// TIA Portal V16 export
// export: Created 2023-03-29T11:03:18.3037804Z, ExportSetting WithDefaults, DisplayName Totally Integrated Automation Portal, DisplayVersion V16 Update 6, DisplayName TIA Portal Version Control Interface, DisplayVersion V16 Update 2, DisplayName TIA Portal Openness, DisplayVersion V16 Update 6, DisplayName STEP 7 Professional, DisplayVersion V16 Update 6, DisplayName STEP 7 Safety, DisplayVersion V16, DisplayName WinCC Advanced, DisplayVersion V16 Update 6
ORGANIZATION_BLOCK "Main"   // OB1, LAD, ProgramCycle
TITLE = "Main Program Sweep (Cycle)"
{ S7_Optimized_Access := 'TRUE' }
VERSION : 0.1
// stored: AutoNumber true, IsIECCheckEnabled false, SetENOAutomatically false
   VAR_INPUT
      Initial_Call : Bool;   // Initial call of this OB
      Remanence : Bool;   // =True, if remanent data are available
   END_VAR
   VAR_TEMP   // added for the SCL form of the ladder/FBD networks
      _w1 : Bool;
      _w2 : Bool;
   END_VAR
BEGIN

REGION Network 1: Diagnostyka przerwań
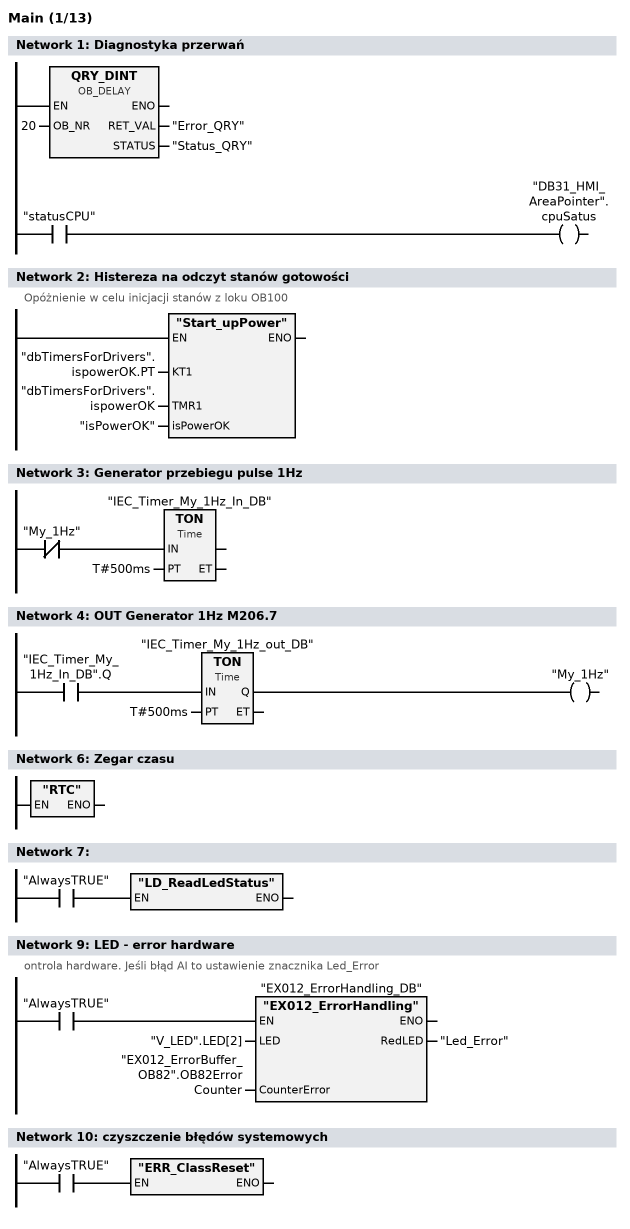
   RUNG wire#powerrail
      { S7_Templates := "obnr_type := OB_DELAY" } QRY_DINT(OB_NR := 20, RET_VAL => "Error_QRY", STATUS => "Status_QRY")
   END_RUNG
   RUNG wire#powerrail
      Contact( "statusCPU" )
      Coil( "DB31_HMI_AreaPointer".cpuSatus )
   END_RUNG
   // the same network as SCL:
   "Error_QRY" := QRY_DINT(OB_NR := 20, STATUS => "Status_QRY");
   "DB31_HMI_AreaPointer".cpuSatus := "statusCPU";
END_REGION

REGION Network 2: Histereza na odczyt stanów gotowości
   // Opóżnienie w celu inicjacji stanów z loku OB100
   RUNG wire#powerrail
      "Start_upPower"(KT1 := "dbTimersForDrivers".ispowerOK.PT, TMR1 := "dbTimersForDrivers".ispowerOK, isPowerOK := "isPowerOK")
   END_RUNG
   // the same network as SCL:
   "Start_upPower"(KT1 := "dbTimersForDrivers".ispowerOK.PT,
                   TMR1 := "dbTimersForDrivers".ispowerOK,
                   isPowerOK := "isPowerOK");
END_REGION

REGION Network 3: Generator przebiegu pulse 1Hz
   RUNG wire#powerrail
      I_Contact( "My_1Hz" )
      { S7_Templates := "time_type := Time" } "IEC_Timer_My_1Hz_In_DB".TON(pt := T#500ms, et =>)
   END_RUNG
   // the same network as SCL:
   "IEC_Timer_My_1Hz_In_DB".TON(IN := NOT "My_1Hz", PT := T#500ms);
END_REGION

REGION Network 4: OUT Generator 1Hz M206.7
   RUNG wire#powerrail
      Contact( "IEC_Timer_My_1Hz_In_DB".Q )
      { S7_Templates := "time_type := Time" } "IEC_Timer_My_1Hz_out_DB".TON(pt := T#500ms, et =>)
      Coil( "My_1Hz" )
   END_RUNG
   // the same network as SCL:
   "IEC_Timer_My_1Hz_out_DB".TON(IN := "IEC_Timer_My_1Hz_In_DB".Q, PT := T#500ms);
   "My_1Hz" := "IEC_Timer_My_1Hz_out_DB".Q;
END_REGION

REGION Network 6: Zegar czasu
   RUNG wire#powerrail
      "RTC"()
   END_RUNG
   // the same network as SCL:
   "RTC"();
END_REGION

REGION Network 7
   RUNG wire#powerrail
      Contact( "AlwaysTRUE" )
      "LD_ReadLedStatus"()
   END_RUNG
   // the same network as SCL:
   IF "AlwaysTRUE" THEN "LD_ReadLedStatus"(); END_IF;
END_REGION

REGION Network 8 (SCL): LED kontrola RUN
   // Przekazanie  stanu LED 1 CPU
   "DB31_HMI_AreaPointer".getPLCMode := "V_LED".LED[1];
END_REGION

REGION Network 9: LED - error hardware
   // ontrola hardware. Jeśli błąd AI to ustawienie znacznika Led_Error
   RUNG wire#powerrail
      Contact( "AlwaysTRUE" )
      "EX012_ErrorHandling_DB"(LED := "V_LED".LED[2], CounterError := "EX012_ErrorBuffer_OB82".OB82ErrorCounter, RedLED => "Led_Error")
   END_RUNG
   // the same network as SCL:
   IF "AlwaysTRUE" THEN
       "EX012_ErrorHandling_DB"(LED := "V_LED".LED[2],   // "EX012_ErrorHandling"
                               CounterError := "EX012_ErrorBuffer_OB82".OB82ErrorCounter,
                               RedLED => "Led_Error");
   END_IF;
END_REGION

REGION Network 10: czyszczenie błędów systemowych
   RUNG wire#powerrail
      Contact( "AlwaysTRUE" )
      "ERR_ClassReset"()
   END_RUNG
   // the same network as SCL:
   IF "AlwaysTRUE" THEN "ERR_ClassReset"(); END_IF;
END_REGION

REGION Network 11: kontrola błedów
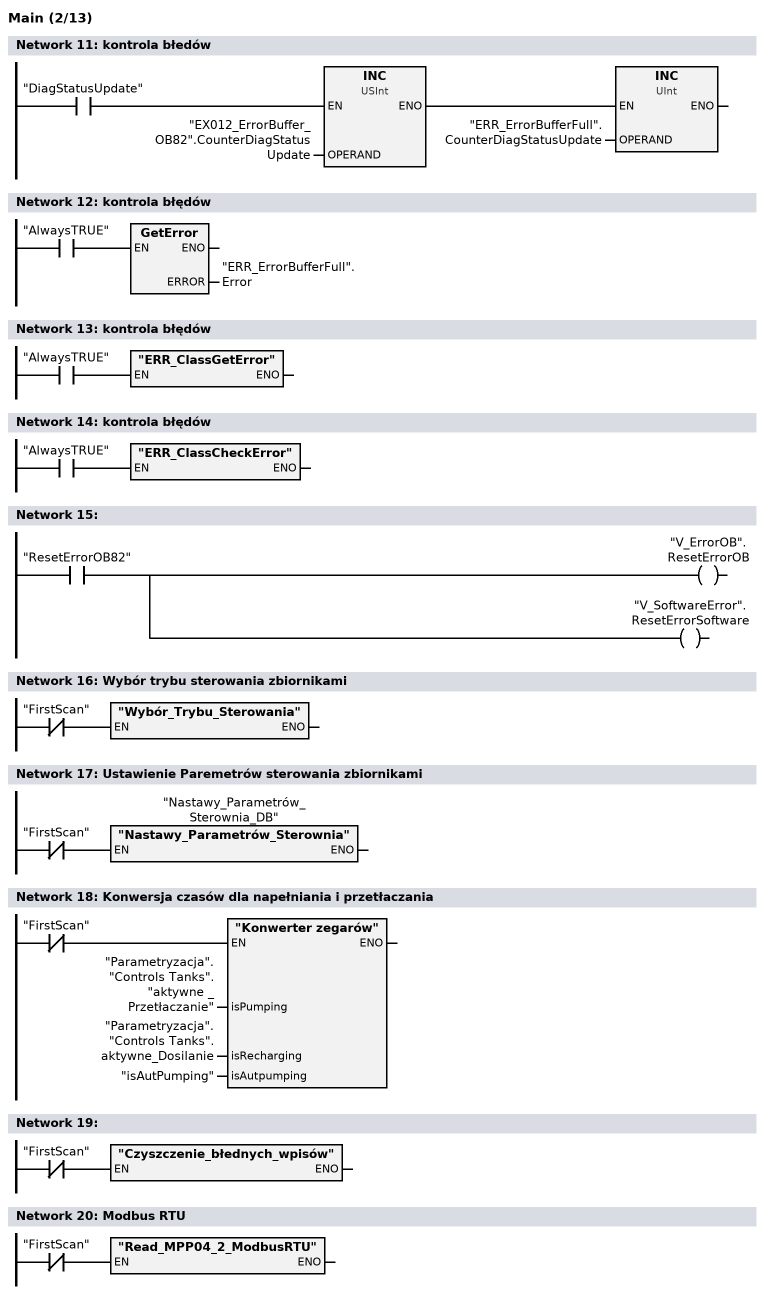
   RUNG wire#powerrail
      Contact( "DiagStatusUpdate" )
      { S7_Templates := "DestType := USInt" } Inc( "EX012_ErrorBuffer_OB82".CounterDiagStatusUpdate )
      { S7_Templates := "DestType := UInt" } Inc( "ERR_ErrorBufferFull".CounterDiagStatusUpdate )
   END_RUNG
   // the same network as SCL:
   IF "DiagStatusUpdate" THEN
       "EX012_ErrorBuffer_OB82".CounterDiagStatusUpdate := "EX012_ErrorBuffer_OB82".CounterDiagStatusUpdate + 1;
       "ERR_ErrorBufferFull".CounterDiagStatusUpdate := "ERR_ErrorBufferFull".CounterDiagStatusUpdate + 1;
   END_IF;
END_REGION

REGION Network 12: kontrola błędów
   // no SCL statement known for GetError: written as a call
   IF "AlwaysTRUE" THEN GetError(error => "ERR_ErrorBufferFull".Error); END_IF;
END_REGION

REGION Network 13: kontrola błędów
   RUNG wire#powerrail
      Contact( "AlwaysTRUE" )
      "ERR_ClassGetError"()
   END_RUNG
   // the same network as SCL:
   IF "AlwaysTRUE" THEN "ERR_ClassGetError"(); END_IF;
END_REGION

REGION Network 14: kontrola błędów
   RUNG wire#powerrail
      Contact( "AlwaysTRUE" )
      "ERR_ClassCheckError"()
   END_RUNG
   // the same network as SCL:
   IF "AlwaysTRUE" THEN "ERR_ClassCheckError"(); END_IF;
END_REGION

REGION Network 15
   RUNG wire#powerrail
      Contact( "ResetErrorOB82" )
      wire#w1
      Coil( "V_ErrorOB".ResetErrorOB )
   END_RUNG
   RUNG wire#w1
      Coil( "V_SoftwareError".ResetErrorSoftware )
   END_RUNG
   // the same network as SCL:
   "V_ErrorOB".ResetErrorOB := "ResetErrorOB82";
   "V_SoftwareError".ResetErrorSoftware := "ResetErrorOB82";
END_REGION

REGION Network 16: Wybór trybu sterowania zbiornikami
   RUNG wire#powerrail
      I_Contact( "FirstScan" )
      "Wybór_Trybu_Sterowania"()
   END_RUNG
   // the same network as SCL:
   IF NOT "FirstScan" THEN "Wybór_Trybu_Sterowania"(); END_IF;
END_REGION

REGION Network 17: Ustawienie Paremetrów sterowania zbiornikami
   RUNG wire#powerrail
      I_Contact( "FirstScan" )
      "Nastawy_Parametrów_Sterownia_DB"()
   END_RUNG
   // the same network as SCL:
   IF NOT "FirstScan" THEN
       "Nastawy_Parametrów_Sterownia_DB"();   // "Nastawy_Parametrów_Sterownia"
   END_IF;
END_REGION

REGION Network 18: Konwersja czasów dla napełniania i przetłaczania
   RUNG wire#powerrail
      I_Contact( "FirstScan" )
      "Konwerter zegarów"(isPumping := "Parametryzacja"."Controls Tanks"."aktywne _Przetłaczanie", isRecharging := "Parametryzacja"."Controls Tanks".aktywne_Dosilanie, isAutpumping := "isAutPumping")
   END_RUNG
   // the same network as SCL:
   IF NOT "FirstScan" THEN
       "Konwerter zegarów"(isPumping := "Parametryzacja"."Controls Tanks"."aktywne _Przetłaczanie",
                           isRecharging := "Parametryzacja"."Controls Tanks".aktywne_Dosilanie,
                           isAutpumping := "isAutPumping");
   END_IF;
END_REGION

REGION Network 19
   RUNG wire#powerrail
      I_Contact( "FirstScan" )
      "Czyszczenie_błednych_wpisów"()
   END_RUNG
   // the same network as SCL:
   IF NOT "FirstScan" THEN "Czyszczenie_błednych_wpisów"(); END_IF;
END_REGION

REGION Network 20: Modbus RTU
   RUNG wire#powerrail
      I_Contact( "FirstScan" )
      "Read_MPP04_2_ModbusRTU"()
   END_RUNG
   // the same network as SCL:
   IF NOT "FirstScan" THEN "Read_MPP04_2_ModbusRTU"(); END_IF;
END_REGION

REGION Network 21: Analogi przekazanie do dbHold Modbus TCP
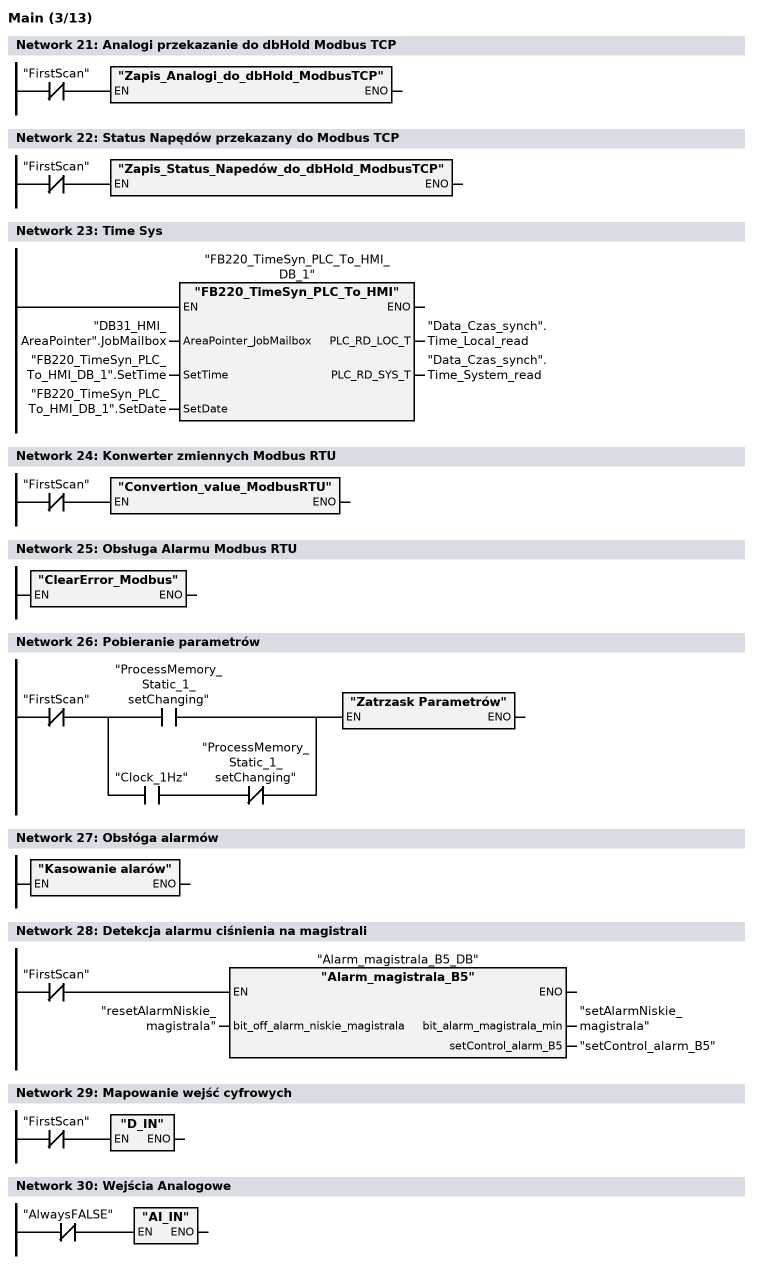
   RUNG wire#powerrail
      I_Contact( "FirstScan" )
      "Zapis_Analogi_do_dbHold_ModbusTCP"()
   END_RUNG
   // the same network as SCL:
   IF NOT "FirstScan" THEN "Zapis_Analogi_do_dbHold_ModbusTCP"(); END_IF;
END_REGION

REGION Network 22: Status Napędów przekazany do Modbus TCP
   RUNG wire#powerrail
      I_Contact( "FirstScan" )
      "Zapis_Status_Napedów_do_dbHold_ModbusTCP"()
   END_RUNG
   // the same network as SCL:
   IF NOT "FirstScan" THEN "Zapis_Status_Napedów_do_dbHold_ModbusTCP"(); END_IF;
END_REGION

REGION Network 23: Time Sys
   RUNG wire#powerrail
      "FB220_TimeSyn_PLC_To_HMI_DB_1"(AreaPointer_JobMailbox := "DB31_HMI_AreaPointer".JobMailbox, SetTime := "FB220_TimeSyn_PLC_To_HMI_DB_1".SetTime, SetDate := "FB220_TimeSyn_PLC_To_HMI_DB_1".SetDate, PLC_RD_LOC_T => "Data_Czas_synch".Time_Local_read, PLC_RD_SYS_T => "Data_Czas_synch".Time_System_read)
   END_RUNG
   // the same network as SCL:
   "FB220_TimeSyn_PLC_To_HMI_DB_1"(AreaPointer_JobMailbox := "DB31_HMI_AreaPointer".JobMailbox,   // "FB220_TimeSyn_PLC_To_HMI"
                           SetTime := "FB220_TimeSyn_PLC_To_HMI_DB_1".SetTime,
                           SetDate := "FB220_TimeSyn_PLC_To_HMI_DB_1".SetDate,
                           PLC_RD_LOC_T => "Data_Czas_synch".Time_Local_read,
                           PLC_RD_SYS_T => "Data_Czas_synch".Time_System_read);
END_REGION

REGION Network 24: Konwerter zmiennych Modbus RTU
   RUNG wire#powerrail
      I_Contact( "FirstScan" )
      "Convertion_value_ModbusRTU"()
   END_RUNG
   // the same network as SCL:
   IF NOT "FirstScan" THEN "Convertion_value_ModbusRTU"(); END_IF;
END_REGION

REGION Network 25: Obsługa Alarmu Modbus RTU
   RUNG wire#powerrail
      "ClearError_Modbus"()
   END_RUNG
   // the same network as SCL:
   "ClearError_Modbus"();
END_REGION

REGION Network 26: Pobieranie parametrów
   RUNG wire#powerrail
      I_Contact( "FirstScan" )
      wire#w1
      Contact( "ProcessMemory_Static_1_setChanging" )
      wire#w2
      "Zatrzask Parametrów"()
   END_RUNG
   RUNG wire#w1
      Contact( "Clock_1Hz" )
      I_Contact( "ProcessMemory_Static_1_setChanging" )
   END_RUNG wire#w2
   // the same network as SCL:
   IF NOT "FirstScan" AND ("ProcessMemory_Static_1_setChanging" OR ("Clock_1Hz" AND NOT "ProcessMemory_Static_1_setChanging")) THEN
       "Zatrzask Parametrów"();
   END_IF;
END_REGION

REGION Network 27: Obsłóga alarmów
   RUNG wire#powerrail
      "Kasowanie alarów"()
   END_RUNG
   // the same network as SCL:
   "Kasowanie alarów"();
END_REGION

REGION Network 28: Detekcja alarmu ciśnienia na magistrali
   RUNG wire#powerrail
      I_Contact( "FirstScan" )
      "Alarm_magistrala_B5_DB"(bit_off_alarm_niskie_magistrala := "resetAlarmNiskie_magistrala", bit_alarm_magistrala_min => "setAlarmNiskie_magistrala", setControl_alarm_B5 => "setControl_alarm_B5")
   END_RUNG
   // the same network as SCL:
   IF NOT "FirstScan" THEN
       "Alarm_magistrala_B5_DB"(bit_off_alarm_niskie_magistrala := "resetAlarmNiskie_magistrala",   // "Alarm_magistrala_B5"
                               bit_alarm_magistrala_min => "setAlarmNiskie_magistrala",
                               setControl_alarm_B5 => "setControl_alarm_B5");
   END_IF;
END_REGION

REGION Network 29: Mapowanie wejść cyfrowych
   RUNG wire#powerrail
      I_Contact( "FirstScan" )
      "D_IN"()
   END_RUNG
   // the same network as SCL:
   IF NOT "FirstScan" THEN "D_IN"(); END_IF;
END_REGION

REGION Network 30: Wejścia Analogowe
   RUNG wire#powerrail
      I_Contact( "AlwaysFALSE" )
      "AI_IN"()
   END_RUNG
   // the same network as SCL:
   IF NOT "AlwaysFALSE" THEN "AI_IN"(); END_IF;
END_REGION

REGION Network 31: Detekcja błędu nadajnika położenia Z10
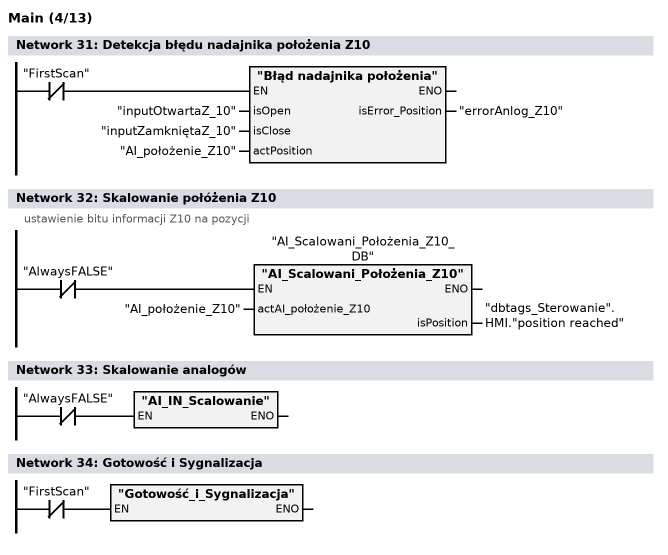
   RUNG wire#powerrail
      I_Contact( "FirstScan" )
      "Błąd nadajnika położenia"(isOpen := "inputOtwartaZ_10", isClose := "inputZamkniętaZ_10", actPosition := "AI_położenie_Z10", isError_Position => "errorAnlog_Z10")
   END_RUNG
   // the same network as SCL:
   IF NOT "FirstScan" THEN
       "Błąd nadajnika położenia"(isOpen := "inputOtwartaZ_10",
                               isClose := "inputZamkniętaZ_10",
                               actPosition := "AI_położenie_Z10",
                               isError_Position => "errorAnlog_Z10");
   END_IF;
END_REGION

REGION Network 32: Skalowanie połóżenia Z10
   // ustawienie bitu informacji Z10 na pozycji
   RUNG wire#powerrail
      I_Contact( "AlwaysFALSE" )
      "AI_Scalowani_Położenia_Z10_DB"(actAI_położenie_Z10 := "AI_położenie_Z10", isPosition => "dbtags_Sterowanie".HMI."position reached")
   END_RUNG
   // the same network as SCL:
   IF NOT "AlwaysFALSE" THEN
       "AI_Scalowani_Położenia_Z10_DB"(actAI_położenie_Z10 := "AI_położenie_Z10",   // "AI_Scalowani_Położenia_Z10"
                               isPosition => "dbtags_Sterowanie".HMI."position reached");
   END_IF;
END_REGION

REGION Network 33: Skalowanie analogów
   RUNG wire#powerrail
      I_Contact( "AlwaysFALSE" )
      "AI_IN_Scalowanie"()
   END_RUNG
   // the same network as SCL:
   IF NOT "AlwaysFALSE" THEN "AI_IN_Scalowanie"(); END_IF;
END_REGION

REGION Network 34: Gotowość i Sygnalizacja
   RUNG wire#powerrail
      I_Contact( "FirstScan" )
      "Gotowość_i_Sygnalizacja"()
   END_RUNG
   // the same network as SCL:
   IF NOT "FirstScan" THEN "Gotowość_i_Sygnalizacja"(); END_IF;
END_REGION

REGION Network 35
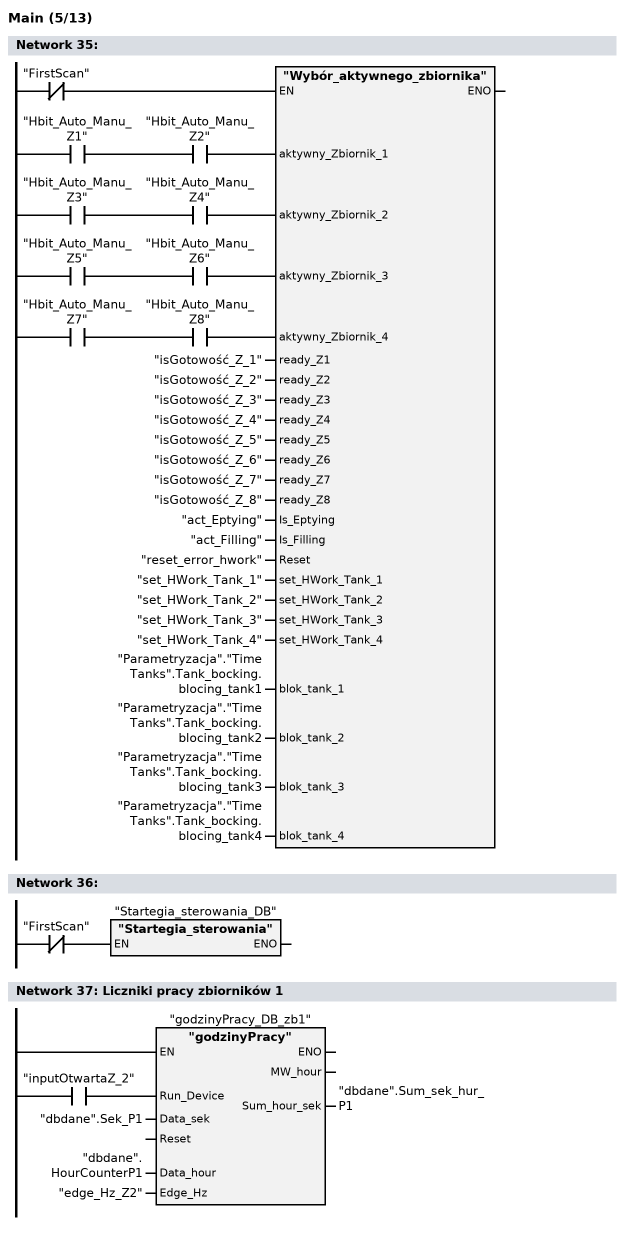
   RUNG wire#powerrail
      I_Contact( "FirstScan" )
      "Wybór_aktywnego_zbiornika"(aktywny_Zbiornik_1 := wire#w1, aktywny_Zbiornik_2 := wire#w2, aktywny_Zbiornik_3 := wire#w3, aktywny_Zbiornik_4 := wire#w4, ready_Z1 := "isGotowość_Z_1", ready_Z2 := "isGotowość_Z_2", ready_Z3 := "isGotowość_Z_3", ready_Z4 := "isGotowość_Z_4", ready_Z5 := "isGotowość_Z_5", ready_Z6 := "isGotowość_Z_6", ready_Z7 := "isGotowość_Z_7", ready_Z8 := "isGotowość_Z_8", Is_Eptying := "act_Eptying", Is_Filling := "act_Filling", Reset := "reset_error_hwork", set_HWork_Tank_1 := "set_HWork_Tank_1", set_HWork_Tank_2 := "set_HWork_Tank_2", set_HWork_Tank_3 := "set_HWork_Tank_3", set_HWork_Tank_4 := "set_HWork_Tank_4", blok_tank_1 := "Parametryzacja"."Time Tanks".Tank_bocking.blocing_tank1, blok_tank_2 := "Parametryzacja"."Time Tanks".Tank_bocking.blocing_tank2, blok_tank_3 := "Parametryzacja"."Time Tanks".Tank_bocking.blocing_tank3, blok_tank_4 := "Parametryzacja"."Time Tanks".Tank_bocking.blocing_tank4)
   END_RUNG
   RUNG wire#powerrail
      Contact( "Hbit_Auto_Manu_Z1" )
      Contact( "Hbit_Auto_Manu_Z2" )
   END_RUNG wire#w1
   RUNG wire#powerrail
      Contact( "Hbit_Auto_Manu_Z3" )
      Contact( "Hbit_Auto_Manu_Z4" )
   END_RUNG wire#w2
   RUNG wire#powerrail
      Contact( "Hbit_Auto_Manu_Z5" )
      Contact( "Hbit_Auto_Manu_Z6" )
   END_RUNG wire#w3
   RUNG wire#powerrail
      Contact( "Hbit_Auto_Manu_Z7" )
      Contact( "Hbit_Auto_Manu_Z8" )
   END_RUNG wire#w4
   // the same network as SCL:
   IF NOT "FirstScan" THEN
       "Wybór_aktywnego_zbiornika"(aktywny_Zbiornik_1 := "Hbit_Auto_Manu_Z1" AND "Hbit_Auto_Manu_Z2",
                               aktywny_Zbiornik_2 := "Hbit_Auto_Manu_Z3" AND "Hbit_Auto_Manu_Z4",
                               aktywny_Zbiornik_3 := "Hbit_Auto_Manu_Z5" AND "Hbit_Auto_Manu_Z6",
                               aktywny_Zbiornik_4 := "Hbit_Auto_Manu_Z7" AND "Hbit_Auto_Manu_Z8",
                               ready_Z1 := "isGotowość_Z_1",
                               ready_Z2 := "isGotowość_Z_2",
                               ready_Z3 := "isGotowość_Z_3",
                               ready_Z4 := "isGotowość_Z_4",
                               ready_Z5 := "isGotowość_Z_5",
                               ready_Z6 := "isGotowość_Z_6",
                               ready_Z7 := "isGotowość_Z_7",
                               ready_Z8 := "isGotowość_Z_8",
                               Is_Eptying := "act_Eptying",
                               Is_Filling := "act_Filling",
                               Reset := "reset_error_hwork",
                               set_HWork_Tank_1 := "set_HWork_Tank_1",
                               set_HWork_Tank_2 := "set_HWork_Tank_2",
                               set_HWork_Tank_3 := "set_HWork_Tank_3",
                               set_HWork_Tank_4 := "set_HWork_Tank_4",
                               blok_tank_1 := "Parametryzacja"."Time Tanks".Tank_bocking.blocing_tank1,
                               blok_tank_2 := "Parametryzacja"."Time Tanks".Tank_bocking.blocing_tank2,
                               blok_tank_3 := "Parametryzacja"."Time Tanks".Tank_bocking.blocing_tank3,
                               blok_tank_4 := "Parametryzacja"."Time Tanks".Tank_bocking.blocing_tank4);
   END_IF;
END_REGION

REGION Network 36
   RUNG wire#powerrail
      I_Contact( "FirstScan" )
      "Startegia_sterowania_DB"()
   END_RUNG
   // the same network as SCL:
   IF NOT "FirstScan" THEN
       "Startegia_sterowania_DB"();   // "Startegia_sterowania"
   END_IF;
END_REGION

REGION Network 37: Liczniki pracy zbiorników 1
   RUNG wire#powerrail
      "godzinyPracy_DB_zb1"(Run_Device := wire#w1, Data_sek := "dbdane".Sek_P1, Reset :=, Data_hour := "dbdane".HourCounterP1, Edge_Hz := "edge_Hz_Z2", MW_hour =>, Sum_hour_sek => "dbdane".Sum_sek_hur_P1)
   END_RUNG
   RUNG wire#powerrail
      Contact( "inputOtwartaZ_2" )
   END_RUNG wire#w1
   // the same network as SCL:
   "godzinyPracy_DB_zb1"(Run_Device := "inputOtwartaZ_2",   // "godzinyPracy"
                         Data_sek := "dbdane".Sek_P1,
                         Data_hour := "dbdane".HourCounterP1,
                         Edge_Hz := "edge_Hz_Z2",
                         Sum_hour_sek => "dbdane".Sum_sek_hur_P1);
END_REGION

REGION Network 38: Liczniki pracy zbiorników 2
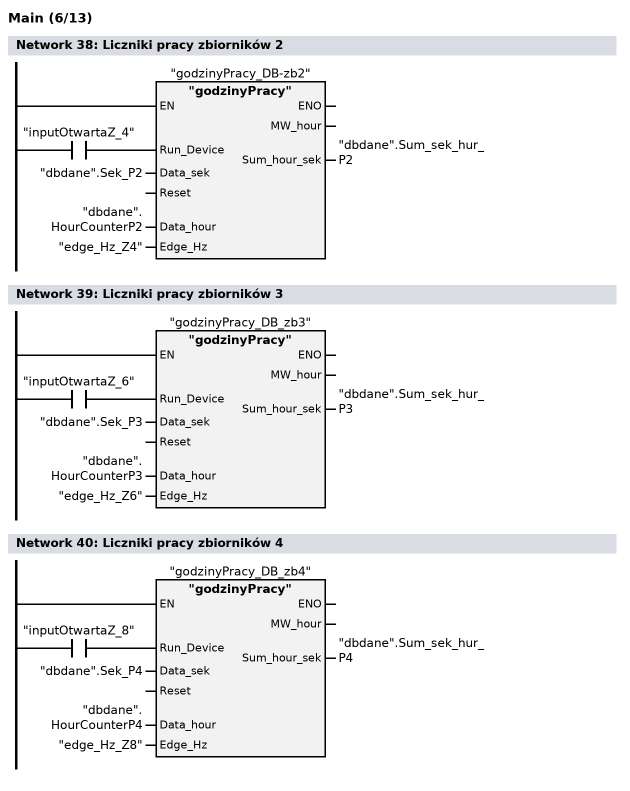
   RUNG wire#powerrail
      "godzinyPracy_DB-zb2"(Run_Device := wire#w1, Data_sek := "dbdane".Sek_P2, Reset :=, Data_hour := "dbdane".HourCounterP2, Edge_Hz := "edge_Hz_Z4", MW_hour =>, Sum_hour_sek => "dbdane".Sum_sek_hur_P2)
   END_RUNG
   RUNG wire#powerrail
      Contact( "inputOtwartaZ_4" )
   END_RUNG wire#w1
   // the same network as SCL:
   "godzinyPracy_DB-zb2"(Run_Device := "inputOtwartaZ_4",   // "godzinyPracy"
                         Data_sek := "dbdane".Sek_P2,
                         Data_hour := "dbdane".HourCounterP2,
                         Edge_Hz := "edge_Hz_Z4",
                         Sum_hour_sek => "dbdane".Sum_sek_hur_P2);
END_REGION

REGION Network 39: Liczniki pracy zbiorników 3
   RUNG wire#powerrail
      "godzinyPracy_DB_zb3"(Run_Device := wire#w1, Data_sek := "dbdane".Sek_P3, Reset :=, Data_hour := "dbdane".HourCounterP3, Edge_Hz := "edge_Hz_Z6", MW_hour =>, Sum_hour_sek => "dbdane".Sum_sek_hur_P3)
   END_RUNG
   RUNG wire#powerrail
      Contact( "inputOtwartaZ_6" )
   END_RUNG wire#w1
   // the same network as SCL:
   "godzinyPracy_DB_zb3"(Run_Device := "inputOtwartaZ_6",   // "godzinyPracy"
                         Data_sek := "dbdane".Sek_P3,
                         Data_hour := "dbdane".HourCounterP3,
                         Edge_Hz := "edge_Hz_Z6",
                         Sum_hour_sek => "dbdane".Sum_sek_hur_P3);
END_REGION

REGION Network 40: Liczniki pracy zbiorników 4
   RUNG wire#powerrail
      "godzinyPracy_DB_zb4"(Run_Device := wire#w1, Data_sek := "dbdane".Sek_P4, Reset :=, Data_hour := "dbdane".HourCounterP4, Edge_Hz := "edge_Hz_Z8", MW_hour =>, Sum_hour_sek => "dbdane".Sum_sek_hur_P4)
   END_RUNG
   RUNG wire#powerrail
      Contact( "inputOtwartaZ_8" )
   END_RUNG wire#w1
   // the same network as SCL:
   "godzinyPracy_DB_zb4"(Run_Device := "inputOtwartaZ_8",   // "godzinyPracy"
                         Data_sek := "dbdane".Sek_P4,
                         Data_hour := "dbdane".HourCounterP4,
                         Edge_Hz := "edge_Hz_Z8",
                         Sum_hour_sek => "dbdane".Sum_sek_hur_P4);
END_REGION

REGION Network 41: Sterowanie zbiornikami nr 1
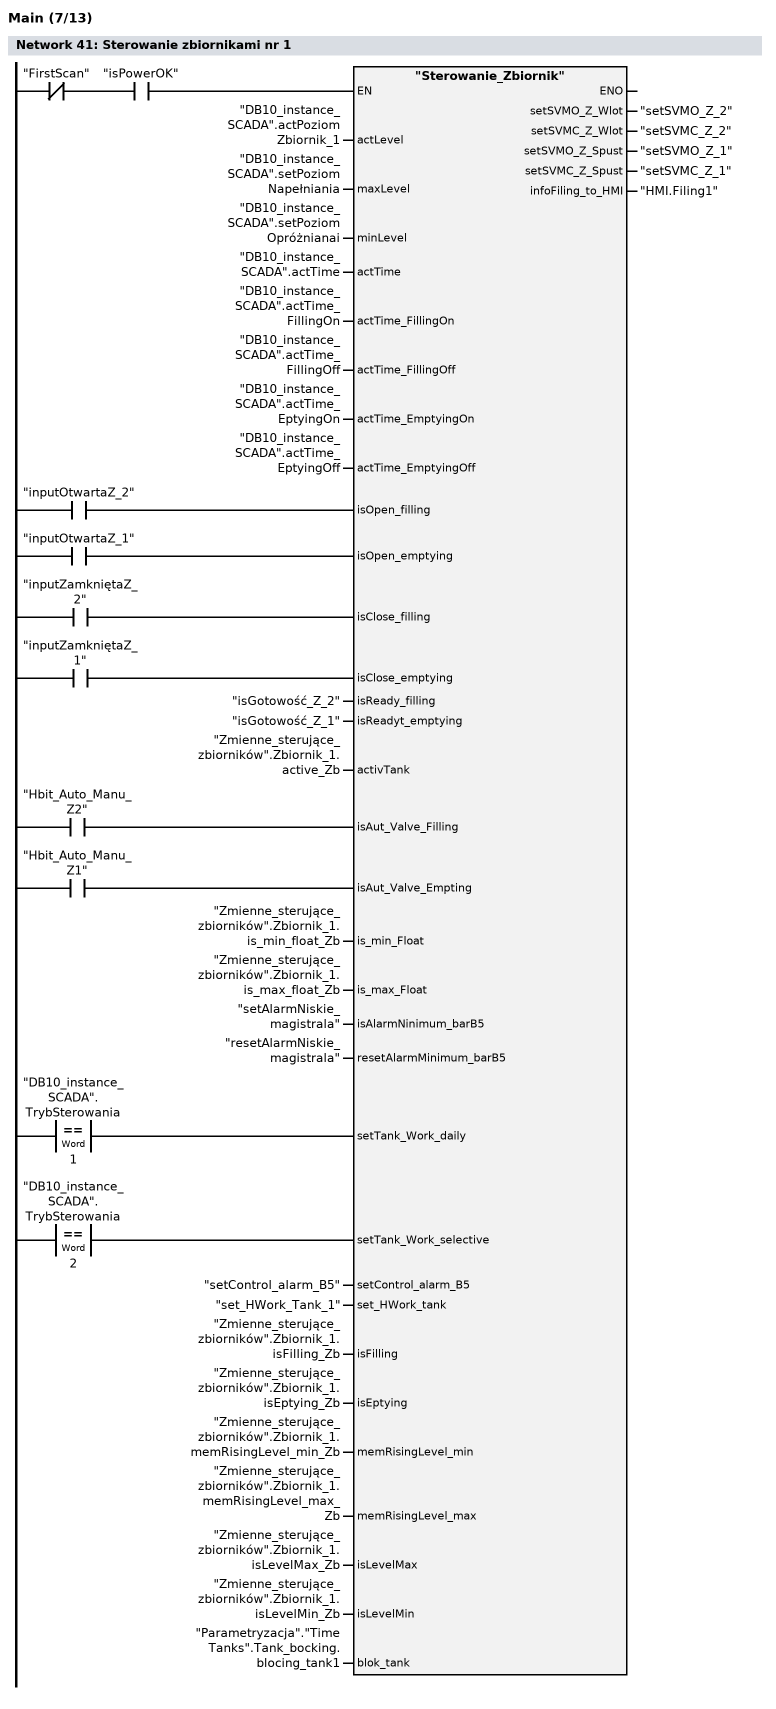
   RUNG wire#powerrail
      I_Contact( "FirstScan" )
      Contact( "isPowerOK" )
      "Sterowanie_Zbiornik"(isOpen_filling := wire#w1, isOpen_emptying := wire#w2, isClose_filling := wire#w3, isClose_emptying := wire#w4, isAut_Valve_Filling := wire#w5, isAut_Valve_Empting := wire#w6, setTank_Work_daily := wire#w7, setTank_Work_selective := wire#w8, actLevel := "DB10_instance_SCADA".actPoziomZbiornik_1, maxLevel := "DB10_instance_SCADA".setPoziomNapełniania, minLevel := "DB10_instance_SCADA".setPoziomOpróżnianai, actTime := "DB10_instance_SCADA".actTime, actTime_FillingOn := "DB10_instance_SCADA".actTime_FillingOn, actTime_FillingOff := "DB10_instance_SCADA".actTime_FillingOff, actTime_EmptyingOn := "DB10_instance_SCADA".actTime_EptyingOn, actTime_EmptyingOff := "DB10_instance_SCADA".actTime_EptyingOff, isReady_filling := "isGotowość_Z_2", isReadyt_emptying := "isGotowość_Z_1", activTank := "Zmienne_sterujące_zbiorników".Zbiornik_1.active_Zb, is_min_Float := "Zmienne_sterujące_zbiorników".Zbiornik_1.is_min_float_Zb, is_max_Float := "Zmienne_sterujące_zbiorników".Zbiornik_1.is_max_float_Zb, isAlarmNinimum_barB5 := "setAlarmNiskie_magistrala", resetAlarmMinimum_barB5 := "resetAlarmNiskie_magistrala", setControl_alarm_B5 := "setControl_alarm_B5", set_HWork_tank := "set_HWork_Tank_1", isFilling := "Zmienne_sterujące_zbiorników".Zbiornik_1.isFilling_Zb, isEptying := "Zmienne_sterujące_zbiorników".Zbiornik_1.isEptying_Zb, memRisingLevel_min := "Zmienne_sterujące_zbiorników".Zbiornik_1.memRisingLevel_min_Zb, memRisingLevel_max := "Zmienne_sterujące_zbiorników".Zbiornik_1.memRisingLevel_max_Zb, isLevelMax := "Zmienne_sterujące_zbiorników".Zbiornik_1.isLevelMax_Zb, isLevelMin := "Zmienne_sterujące_zbiorników".Zbiornik_1.isLevelMin_Zb, blok_tank := "Parametryzacja"."Time Tanks".Tank_bocking.blocing_tank1, setSVMO_Z_Wlot => "setSVMO_Z_2", setSVMC_Z_Wlot => "setSVMC_Z_2", setSVMO_Z_Spust => "setSVMO_Z_1", setSVMC_Z_Spust => "setSVMC_Z_1", infoFiling_to_HMI => "HMI.Filing1")
   END_RUNG
   RUNG wire#powerrail
      Contact( "inputOtwartaZ_2" )
   END_RUNG wire#w1
   RUNG wire#powerrail
      Contact( "inputOtwartaZ_1" )
   END_RUNG wire#w2
   RUNG wire#powerrail
      Contact( "inputZamkniętaZ_2" )
   END_RUNG wire#w3
   RUNG wire#powerrail
      Contact( "inputZamkniętaZ_1" )
   END_RUNG wire#w4
   RUNG wire#powerrail
      Contact( "Hbit_Auto_Manu_Z2" )
   END_RUNG wire#w5
   RUNG wire#powerrail
      Contact( "Hbit_Auto_Manu_Z1" )
   END_RUNG wire#w6
   RUNG wire#powerrail
      { S7_Templates := "SrcType := Word" } EQ_Contact(in1 := "DB10_instance_SCADA".TrybSterowania, in2 := 1)
   END_RUNG wire#w7
   RUNG wire#powerrail
      { S7_Templates := "SrcType := Word" } EQ_Contact(in1 := "DB10_instance_SCADA".TrybSterowania, in2 := 2)
   END_RUNG wire#w8
   // the same network as SCL:
   IF NOT "FirstScan" AND "isPowerOK" THEN
       "Sterowanie_Zbiornik"(actLevel := "DB10_instance_SCADA".actPoziomZbiornik_1,
                             maxLevel := "DB10_instance_SCADA".setPoziomNapełniania,
                             minLevel := "DB10_instance_SCADA".setPoziomOpróżnianai,
                             actTime := "DB10_instance_SCADA".actTime,
                             actTime_FillingOn := "DB10_instance_SCADA".actTime_FillingOn,
                             actTime_FillingOff := "DB10_instance_SCADA".actTime_FillingOff,
                             actTime_EmptyingOn := "DB10_instance_SCADA".actTime_EptyingOn,
                             actTime_EmptyingOff := "DB10_instance_SCADA".actTime_EptyingOff,
                             isOpen_filling := "inputOtwartaZ_2",
                             isOpen_emptying := "inputOtwartaZ_1",
                             isClose_filling := "inputZamkniętaZ_2",
                             isClose_emptying := "inputZamkniętaZ_1",
                             isReady_filling := "isGotowość_Z_2",
                             isReadyt_emptying := "isGotowość_Z_1",
                             activTank := "Zmienne_sterujące_zbiorników".Zbiornik_1.active_Zb,
                             isAut_Valve_Filling := "Hbit_Auto_Manu_Z2",
                             isAut_Valve_Empting := "Hbit_Auto_Manu_Z1",
                             is_min_Float := "Zmienne_sterujące_zbiorników".Zbiornik_1.is_min_float_Zb,
                             is_max_Float := "Zmienne_sterujące_zbiorników".Zbiornik_1.is_max_float_Zb,
                             isAlarmNinimum_barB5 := "setAlarmNiskie_magistrala",
                             resetAlarmMinimum_barB5 := "resetAlarmNiskie_magistrala",
                             setTank_Work_daily := "DB10_instance_SCADA".TrybSterowania = 1,
                             setTank_Work_selective := "DB10_instance_SCADA".TrybSterowania = 2,
                             setControl_alarm_B5 := "setControl_alarm_B5",
                             set_HWork_tank := "set_HWork_Tank_1",
                             isFilling := "Zmienne_sterujące_zbiorników".Zbiornik_1.isFilling_Zb,
                             isEptying := "Zmienne_sterujące_zbiorników".Zbiornik_1.isEptying_Zb,
                             memRisingLevel_min := "Zmienne_sterujące_zbiorników".Zbiornik_1.memRisingLevel_min_Zb,
                             memRisingLevel_max := "Zmienne_sterujące_zbiorników".Zbiornik_1.memRisingLevel_max_Zb,
                             isLevelMax := "Zmienne_sterujące_zbiorników".Zbiornik_1.isLevelMax_Zb,
                             isLevelMin := "Zmienne_sterujące_zbiorników".Zbiornik_1.isLevelMin_Zb,
                             blok_tank := "Parametryzacja"."Time Tanks".Tank_bocking.blocing_tank1,
                             setSVMO_Z_Wlot => "setSVMO_Z_2",
                             setSVMC_Z_Wlot => "setSVMC_Z_2",
                             setSVMO_Z_Spust => "setSVMO_Z_1",
                             setSVMC_Z_Spust => "setSVMC_Z_1",
                             infoFiling_to_HMI => "HMI.Filing1");
   END_IF;
END_REGION

REGION Network 42: Sterowanie zbiornikami nr 2
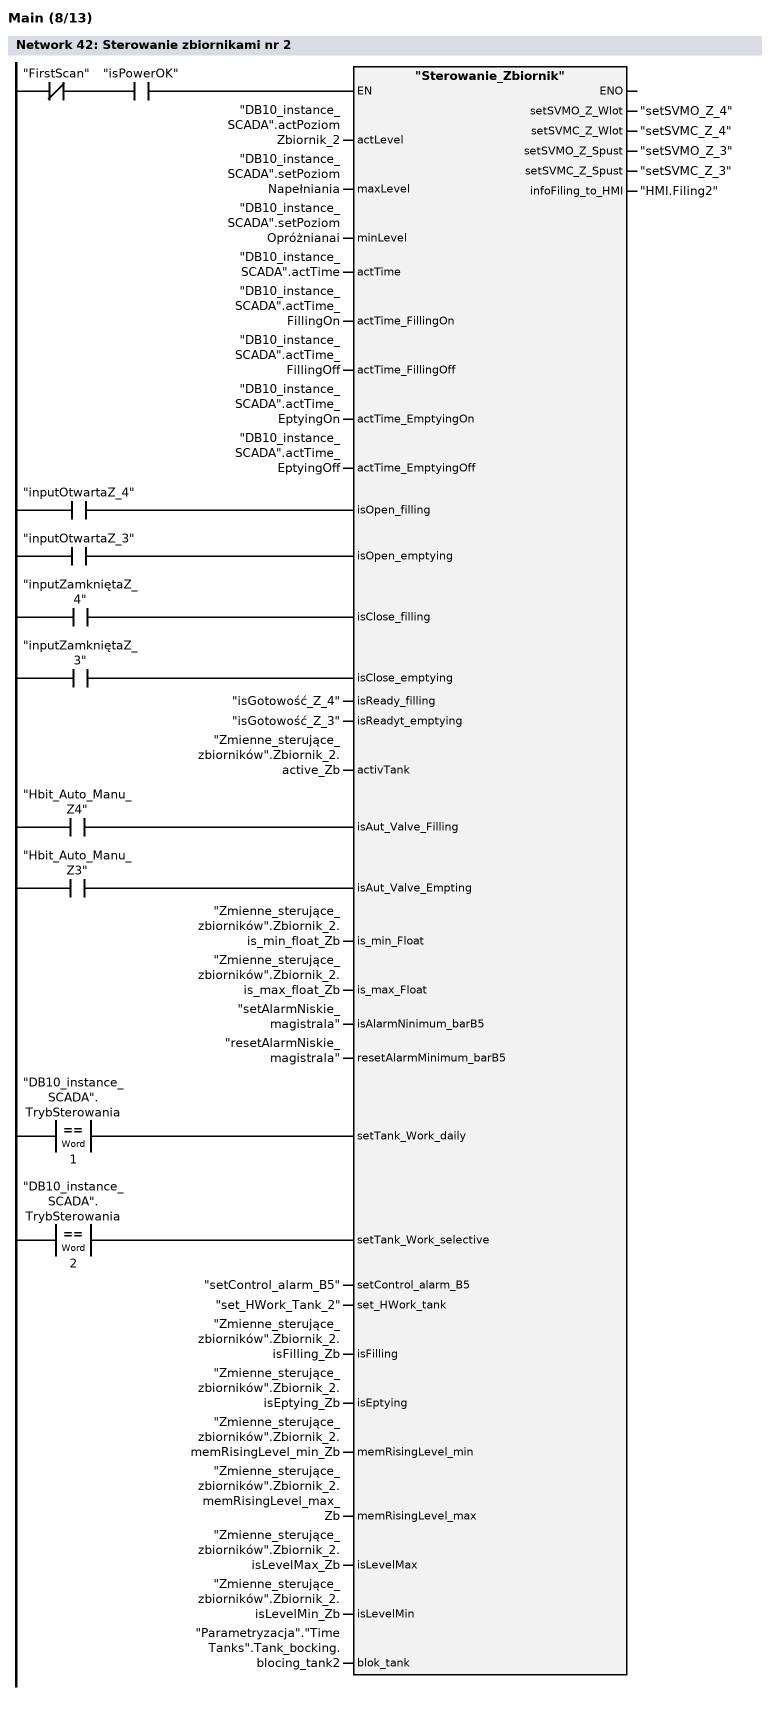
   RUNG wire#powerrail
      I_Contact( "FirstScan" )
      Contact( "isPowerOK" )
      "Sterowanie_Zbiornik"(isOpen_filling := wire#w1, isOpen_emptying := wire#w2, isClose_filling := wire#w3, isClose_emptying := wire#w4, isAut_Valve_Filling := wire#w5, isAut_Valve_Empting := wire#w6, setTank_Work_daily := wire#w7, setTank_Work_selective := wire#w8, actLevel := "DB10_instance_SCADA".actPoziomZbiornik_2, maxLevel := "DB10_instance_SCADA".setPoziomNapełniania, minLevel := "DB10_instance_SCADA".setPoziomOpróżnianai, actTime := "DB10_instance_SCADA".actTime, actTime_FillingOn := "DB10_instance_SCADA".actTime_FillingOn, actTime_FillingOff := "DB10_instance_SCADA".actTime_FillingOff, actTime_EmptyingOn := "DB10_instance_SCADA".actTime_EptyingOn, actTime_EmptyingOff := "DB10_instance_SCADA".actTime_EptyingOff, isReady_filling := "isGotowość_Z_4", isReadyt_emptying := "isGotowość_Z_3", activTank := "Zmienne_sterujące_zbiorników".Zbiornik_2.active_Zb, is_min_Float := "Zmienne_sterujące_zbiorników".Zbiornik_2.is_min_float_Zb, is_max_Float := "Zmienne_sterujące_zbiorników".Zbiornik_2.is_max_float_Zb, isAlarmNinimum_barB5 := "setAlarmNiskie_magistrala", resetAlarmMinimum_barB5 := "resetAlarmNiskie_magistrala", setControl_alarm_B5 := "setControl_alarm_B5", set_HWork_tank := "set_HWork_Tank_2", isFilling := "Zmienne_sterujące_zbiorników".Zbiornik_2.isFilling_Zb, isEptying := "Zmienne_sterujące_zbiorników".Zbiornik_2.isEptying_Zb, memRisingLevel_min := "Zmienne_sterujące_zbiorników".Zbiornik_2.memRisingLevel_min_Zb, memRisingLevel_max := "Zmienne_sterujące_zbiorników".Zbiornik_2.memRisingLevel_max_Zb, isLevelMax := "Zmienne_sterujące_zbiorników".Zbiornik_2.isLevelMax_Zb, isLevelMin := "Zmienne_sterujące_zbiorników".Zbiornik_2.isLevelMin_Zb, blok_tank := "Parametryzacja"."Time Tanks".Tank_bocking.blocing_tank2, setSVMO_Z_Wlot => "setSVMO_Z_4", setSVMC_Z_Wlot => "setSVMC_Z_4", setSVMO_Z_Spust => "setSVMO_Z_3", setSVMC_Z_Spust => "setSVMC_Z_3", infoFiling_to_HMI => "HMI.Filing2")
   END_RUNG
   RUNG wire#powerrail
      Contact( "inputOtwartaZ_4" )
   END_RUNG wire#w1
   RUNG wire#powerrail
      Contact( "inputOtwartaZ_3" )
   END_RUNG wire#w2
   RUNG wire#powerrail
      Contact( "inputZamkniętaZ_4" )
   END_RUNG wire#w3
   RUNG wire#powerrail
      Contact( "inputZamkniętaZ_3" )
   END_RUNG wire#w4
   RUNG wire#powerrail
      Contact( "Hbit_Auto_Manu_Z4" )
   END_RUNG wire#w5
   RUNG wire#powerrail
      Contact( "Hbit_Auto_Manu_Z3" )
   END_RUNG wire#w6
   RUNG wire#powerrail
      { S7_Templates := "SrcType := Word" } EQ_Contact(in1 := "DB10_instance_SCADA".TrybSterowania, in2 := 1)
   END_RUNG wire#w7
   RUNG wire#powerrail
      { S7_Templates := "SrcType := Word" } EQ_Contact(in1 := "DB10_instance_SCADA".TrybSterowania, in2 := 2)
   END_RUNG wire#w8
   // the same network as SCL:
   IF NOT "FirstScan" AND "isPowerOK" THEN
       "Sterowanie_Zbiornik"(actLevel := "DB10_instance_SCADA".actPoziomZbiornik_2,
                             maxLevel := "DB10_instance_SCADA".setPoziomNapełniania,
                             minLevel := "DB10_instance_SCADA".setPoziomOpróżnianai,
                             actTime := "DB10_instance_SCADA".actTime,
                             actTime_FillingOn := "DB10_instance_SCADA".actTime_FillingOn,
                             actTime_FillingOff := "DB10_instance_SCADA".actTime_FillingOff,
                             actTime_EmptyingOn := "DB10_instance_SCADA".actTime_EptyingOn,
                             actTime_EmptyingOff := "DB10_instance_SCADA".actTime_EptyingOff,
                             isOpen_filling := "inputOtwartaZ_4",
                             isOpen_emptying := "inputOtwartaZ_3",
                             isClose_filling := "inputZamkniętaZ_4",
                             isClose_emptying := "inputZamkniętaZ_3",
                             isReady_filling := "isGotowość_Z_4",
                             isReadyt_emptying := "isGotowość_Z_3",
                             activTank := "Zmienne_sterujące_zbiorników".Zbiornik_2.active_Zb,
                             isAut_Valve_Filling := "Hbit_Auto_Manu_Z4",
                             isAut_Valve_Empting := "Hbit_Auto_Manu_Z3",
                             is_min_Float := "Zmienne_sterujące_zbiorników".Zbiornik_2.is_min_float_Zb,
                             is_max_Float := "Zmienne_sterujące_zbiorników".Zbiornik_2.is_max_float_Zb,
                             isAlarmNinimum_barB5 := "setAlarmNiskie_magistrala",
                             resetAlarmMinimum_barB5 := "resetAlarmNiskie_magistrala",
                             setTank_Work_daily := "DB10_instance_SCADA".TrybSterowania = 1,
                             setTank_Work_selective := "DB10_instance_SCADA".TrybSterowania = 2,
                             setControl_alarm_B5 := "setControl_alarm_B5",
                             set_HWork_tank := "set_HWork_Tank_2",
                             isFilling := "Zmienne_sterujące_zbiorników".Zbiornik_2.isFilling_Zb,
                             isEptying := "Zmienne_sterujące_zbiorników".Zbiornik_2.isEptying_Zb,
                             memRisingLevel_min := "Zmienne_sterujące_zbiorników".Zbiornik_2.memRisingLevel_min_Zb,
                             memRisingLevel_max := "Zmienne_sterujące_zbiorników".Zbiornik_2.memRisingLevel_max_Zb,
                             isLevelMax := "Zmienne_sterujące_zbiorników".Zbiornik_2.isLevelMax_Zb,
                             isLevelMin := "Zmienne_sterujące_zbiorników".Zbiornik_2.isLevelMin_Zb,
                             blok_tank := "Parametryzacja"."Time Tanks".Tank_bocking.blocing_tank2,
                             setSVMO_Z_Wlot => "setSVMO_Z_4",
                             setSVMC_Z_Wlot => "setSVMC_Z_4",
                             setSVMO_Z_Spust => "setSVMO_Z_3",
                             setSVMC_Z_Spust => "setSVMC_Z_3",
                             infoFiling_to_HMI => "HMI.Filing2");
   END_IF;
END_REGION

REGION Network 43: Sterowanie zbiornikami nr 3
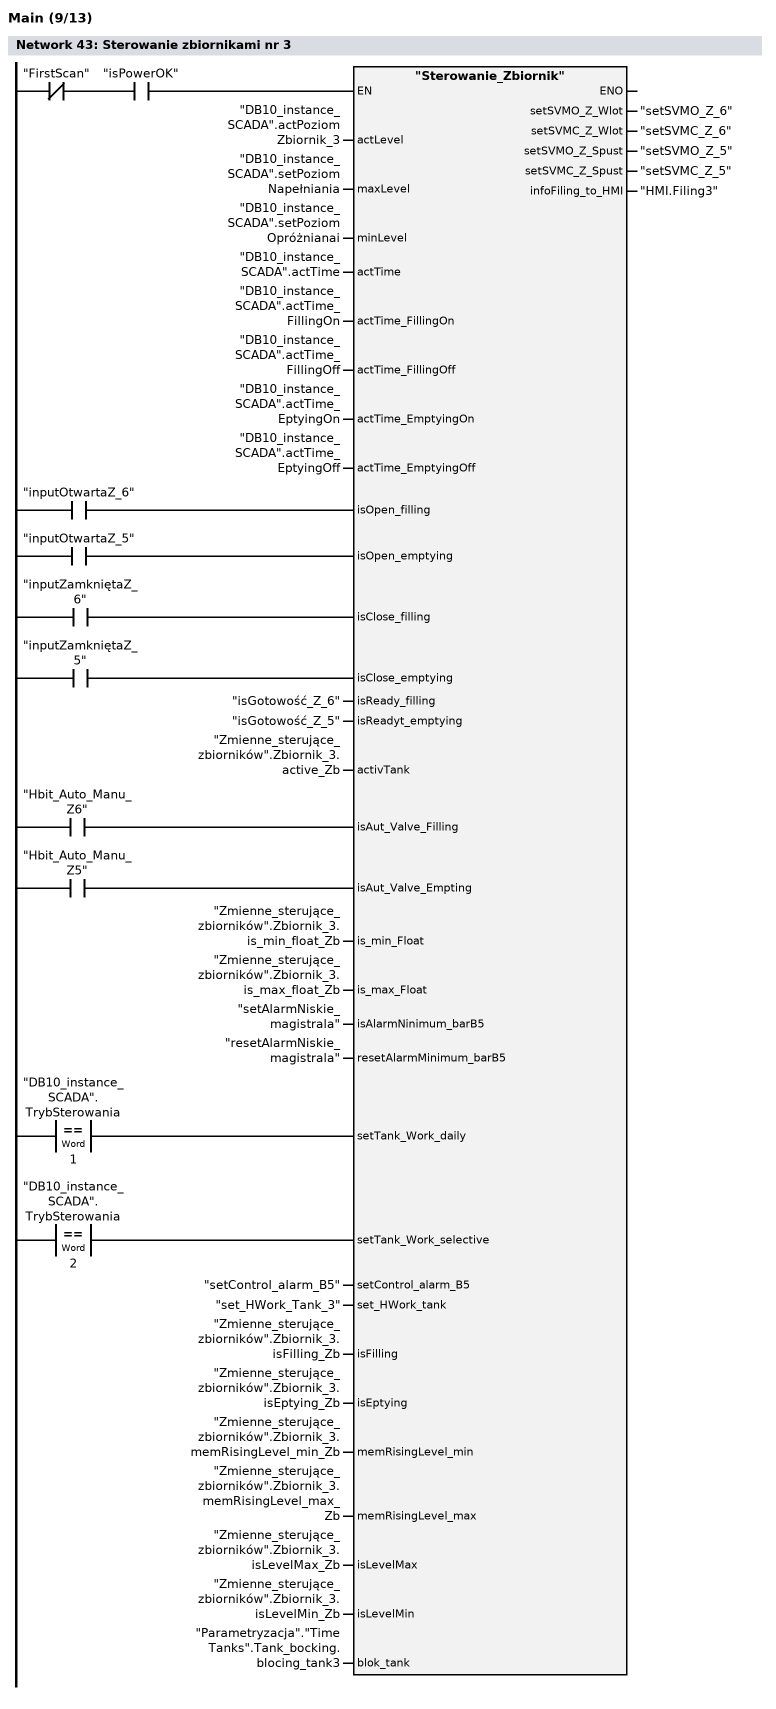
   RUNG wire#powerrail
      I_Contact( "FirstScan" )
      Contact( "isPowerOK" )
      "Sterowanie_Zbiornik"(isOpen_filling := wire#w1, isOpen_emptying := wire#w2, isClose_filling := wire#w3, isClose_emptying := wire#w4, isAut_Valve_Filling := wire#w5, isAut_Valve_Empting := wire#w6, setTank_Work_daily := wire#w7, setTank_Work_selective := wire#w8, actLevel := "DB10_instance_SCADA".actPoziomZbiornik_3, maxLevel := "DB10_instance_SCADA".setPoziomNapełniania, minLevel := "DB10_instance_SCADA".setPoziomOpróżnianai, actTime := "DB10_instance_SCADA".actTime, actTime_FillingOn := "DB10_instance_SCADA".actTime_FillingOn, actTime_FillingOff := "DB10_instance_SCADA".actTime_FillingOff, actTime_EmptyingOn := "DB10_instance_SCADA".actTime_EptyingOn, actTime_EmptyingOff := "DB10_instance_SCADA".actTime_EptyingOff, isReady_filling := "isGotowość_Z_6", isReadyt_emptying := "isGotowość_Z_5", activTank := "Zmienne_sterujące_zbiorników".Zbiornik_3.active_Zb, is_min_Float := "Zmienne_sterujące_zbiorników".Zbiornik_3.is_min_float_Zb, is_max_Float := "Zmienne_sterujące_zbiorników".Zbiornik_3.is_max_float_Zb, isAlarmNinimum_barB5 := "setAlarmNiskie_magistrala", resetAlarmMinimum_barB5 := "resetAlarmNiskie_magistrala", setControl_alarm_B5 := "setControl_alarm_B5", set_HWork_tank := "set_HWork_Tank_3", isFilling := "Zmienne_sterujące_zbiorników".Zbiornik_3.isFilling_Zb, isEptying := "Zmienne_sterujące_zbiorników".Zbiornik_3.isEptying_Zb, memRisingLevel_min := "Zmienne_sterujące_zbiorników".Zbiornik_3.memRisingLevel_min_Zb, memRisingLevel_max := "Zmienne_sterujące_zbiorników".Zbiornik_3.memRisingLevel_max_Zb, isLevelMax := "Zmienne_sterujące_zbiorników".Zbiornik_3.isLevelMax_Zb, isLevelMin := "Zmienne_sterujące_zbiorników".Zbiornik_3.isLevelMin_Zb, blok_tank := "Parametryzacja"."Time Tanks".Tank_bocking.blocing_tank3, setSVMO_Z_Wlot => "setSVMO_Z_6", setSVMC_Z_Wlot => "setSVMC_Z_6", setSVMO_Z_Spust => "setSVMO_Z_5", setSVMC_Z_Spust => "setSVMC_Z_5", infoFiling_to_HMI => "HMI.Filing3")
   END_RUNG
   RUNG wire#powerrail
      Contact( "inputOtwartaZ_6" )
   END_RUNG wire#w1
   RUNG wire#powerrail
      Contact( "inputOtwartaZ_5" )
   END_RUNG wire#w2
   RUNG wire#powerrail
      Contact( "inputZamkniętaZ_6" )
   END_RUNG wire#w3
   RUNG wire#powerrail
      Contact( "inputZamkniętaZ_5" )
   END_RUNG wire#w4
   RUNG wire#powerrail
      Contact( "Hbit_Auto_Manu_Z6" )
   END_RUNG wire#w5
   RUNG wire#powerrail
      Contact( "Hbit_Auto_Manu_Z5" )
   END_RUNG wire#w6
   RUNG wire#powerrail
      { S7_Templates := "SrcType := Word" } EQ_Contact(in1 := "DB10_instance_SCADA".TrybSterowania, in2 := 1)
   END_RUNG wire#w7
   RUNG wire#powerrail
      { S7_Templates := "SrcType := Word" } EQ_Contact(in1 := "DB10_instance_SCADA".TrybSterowania, in2 := 2)
   END_RUNG wire#w8
   // the same network as SCL:
   IF NOT "FirstScan" AND "isPowerOK" THEN
       "Sterowanie_Zbiornik"(actLevel := "DB10_instance_SCADA".actPoziomZbiornik_3,
                             maxLevel := "DB10_instance_SCADA".setPoziomNapełniania,
                             minLevel := "DB10_instance_SCADA".setPoziomOpróżnianai,
                             actTime := "DB10_instance_SCADA".actTime,
                             actTime_FillingOn := "DB10_instance_SCADA".actTime_FillingOn,
                             actTime_FillingOff := "DB10_instance_SCADA".actTime_FillingOff,
                             actTime_EmptyingOn := "DB10_instance_SCADA".actTime_EptyingOn,
                             actTime_EmptyingOff := "DB10_instance_SCADA".actTime_EptyingOff,
                             isOpen_filling := "inputOtwartaZ_6",
                             isOpen_emptying := "inputOtwartaZ_5",
                             isClose_filling := "inputZamkniętaZ_6",
                             isClose_emptying := "inputZamkniętaZ_5",
                             isReady_filling := "isGotowość_Z_6",
                             isReadyt_emptying := "isGotowość_Z_5",
                             activTank := "Zmienne_sterujące_zbiorników".Zbiornik_3.active_Zb,
                             isAut_Valve_Filling := "Hbit_Auto_Manu_Z6",
                             isAut_Valve_Empting := "Hbit_Auto_Manu_Z5",
                             is_min_Float := "Zmienne_sterujące_zbiorników".Zbiornik_3.is_min_float_Zb,
                             is_max_Float := "Zmienne_sterujące_zbiorników".Zbiornik_3.is_max_float_Zb,
                             isAlarmNinimum_barB5 := "setAlarmNiskie_magistrala",
                             resetAlarmMinimum_barB5 := "resetAlarmNiskie_magistrala",
                             setTank_Work_daily := "DB10_instance_SCADA".TrybSterowania = 1,
                             setTank_Work_selective := "DB10_instance_SCADA".TrybSterowania = 2,
                             setControl_alarm_B5 := "setControl_alarm_B5",
                             set_HWork_tank := "set_HWork_Tank_3",
                             isFilling := "Zmienne_sterujące_zbiorników".Zbiornik_3.isFilling_Zb,
                             isEptying := "Zmienne_sterujące_zbiorników".Zbiornik_3.isEptying_Zb,
                             memRisingLevel_min := "Zmienne_sterujące_zbiorników".Zbiornik_3.memRisingLevel_min_Zb,
                             memRisingLevel_max := "Zmienne_sterujące_zbiorników".Zbiornik_3.memRisingLevel_max_Zb,
                             isLevelMax := "Zmienne_sterujące_zbiorników".Zbiornik_3.isLevelMax_Zb,
                             isLevelMin := "Zmienne_sterujące_zbiorników".Zbiornik_3.isLevelMin_Zb,
                             blok_tank := "Parametryzacja"."Time Tanks".Tank_bocking.blocing_tank3,
                             setSVMO_Z_Wlot => "setSVMO_Z_6",
                             setSVMC_Z_Wlot => "setSVMC_Z_6",
                             setSVMO_Z_Spust => "setSVMO_Z_5",
                             setSVMC_Z_Spust => "setSVMC_Z_5",
                             infoFiling_to_HMI => "HMI.Filing3");
   END_IF;
END_REGION

REGION Network 44: Sterowanie zbiornikami nr 4
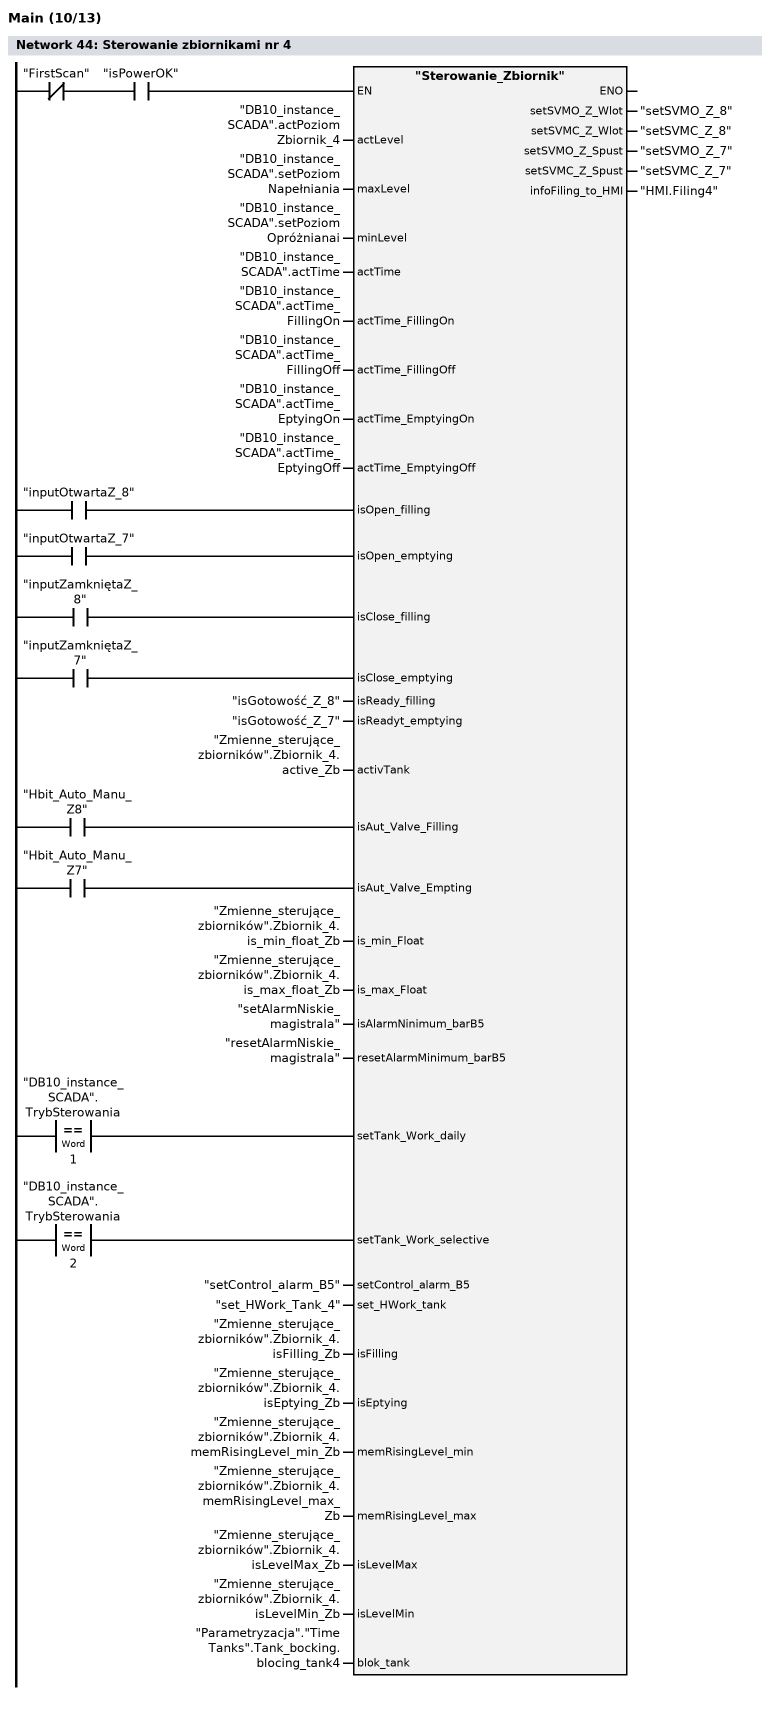
   RUNG wire#powerrail
      I_Contact( "FirstScan" )
      Contact( "isPowerOK" )
      "Sterowanie_Zbiornik"(isOpen_filling := wire#w1, isOpen_emptying := wire#w2, isClose_filling := wire#w3, isClose_emptying := wire#w4, isAut_Valve_Filling := wire#w5, isAut_Valve_Empting := wire#w6, setTank_Work_daily := wire#w7, setTank_Work_selective := wire#w8, actLevel := "DB10_instance_SCADA".actPoziomZbiornik_4, maxLevel := "DB10_instance_SCADA".setPoziomNapełniania, minLevel := "DB10_instance_SCADA".setPoziomOpróżnianai, actTime := "DB10_instance_SCADA".actTime, actTime_FillingOn := "DB10_instance_SCADA".actTime_FillingOn, actTime_FillingOff := "DB10_instance_SCADA".actTime_FillingOff, actTime_EmptyingOn := "DB10_instance_SCADA".actTime_EptyingOn, actTime_EmptyingOff := "DB10_instance_SCADA".actTime_EptyingOff, isReady_filling := "isGotowość_Z_8", isReadyt_emptying := "isGotowość_Z_7", activTank := "Zmienne_sterujące_zbiorników".Zbiornik_4.active_Zb, is_min_Float := "Zmienne_sterujące_zbiorników".Zbiornik_4.is_min_float_Zb, is_max_Float := "Zmienne_sterujące_zbiorników".Zbiornik_4.is_max_float_Zb, isAlarmNinimum_barB5 := "setAlarmNiskie_magistrala", resetAlarmMinimum_barB5 := "resetAlarmNiskie_magistrala", setControl_alarm_B5 := "setControl_alarm_B5", set_HWork_tank := "set_HWork_Tank_4", isFilling := "Zmienne_sterujące_zbiorników".Zbiornik_4.isFilling_Zb, isEptying := "Zmienne_sterujące_zbiorników".Zbiornik_4.isEptying_Zb, memRisingLevel_min := "Zmienne_sterujące_zbiorników".Zbiornik_4.memRisingLevel_min_Zb, memRisingLevel_max := "Zmienne_sterujące_zbiorników".Zbiornik_4.memRisingLevel_max_Zb, isLevelMax := "Zmienne_sterujące_zbiorników".Zbiornik_4.isLevelMax_Zb, isLevelMin := "Zmienne_sterujące_zbiorników".Zbiornik_4.isLevelMin_Zb, blok_tank := "Parametryzacja"."Time Tanks".Tank_bocking.blocing_tank4, setSVMO_Z_Wlot => "setSVMO_Z_8", setSVMC_Z_Wlot => "setSVMC_Z_8", setSVMO_Z_Spust => "setSVMO_Z_7", setSVMC_Z_Spust => "setSVMC_Z_7", infoFiling_to_HMI => "HMI.Filing4")
   END_RUNG
   RUNG wire#powerrail
      Contact( "inputOtwartaZ_8" )
   END_RUNG wire#w1
   RUNG wire#powerrail
      Contact( "inputOtwartaZ_7" )
   END_RUNG wire#w2
   RUNG wire#powerrail
      Contact( "inputZamkniętaZ_8" )
   END_RUNG wire#w3
   RUNG wire#powerrail
      Contact( "inputZamkniętaZ_7" )
   END_RUNG wire#w4
   RUNG wire#powerrail
      Contact( "Hbit_Auto_Manu_Z8" )
   END_RUNG wire#w5
   RUNG wire#powerrail
      Contact( "Hbit_Auto_Manu_Z7" )
   END_RUNG wire#w6
   RUNG wire#powerrail
      { S7_Templates := "SrcType := Word" } EQ_Contact(in1 := "DB10_instance_SCADA".TrybSterowania, in2 := 1)
   END_RUNG wire#w7
   RUNG wire#powerrail
      { S7_Templates := "SrcType := Word" } EQ_Contact(in1 := "DB10_instance_SCADA".TrybSterowania, in2 := 2)
   END_RUNG wire#w8
   // the same network as SCL:
   IF NOT "FirstScan" AND "isPowerOK" THEN
       "Sterowanie_Zbiornik"(actLevel := "DB10_instance_SCADA".actPoziomZbiornik_4,
                             maxLevel := "DB10_instance_SCADA".setPoziomNapełniania,
                             minLevel := "DB10_instance_SCADA".setPoziomOpróżnianai,
                             actTime := "DB10_instance_SCADA".actTime,
                             actTime_FillingOn := "DB10_instance_SCADA".actTime_FillingOn,
                             actTime_FillingOff := "DB10_instance_SCADA".actTime_FillingOff,
                             actTime_EmptyingOn := "DB10_instance_SCADA".actTime_EptyingOn,
                             actTime_EmptyingOff := "DB10_instance_SCADA".actTime_EptyingOff,
                             isOpen_filling := "inputOtwartaZ_8",
                             isOpen_emptying := "inputOtwartaZ_7",
                             isClose_filling := "inputZamkniętaZ_8",
                             isClose_emptying := "inputZamkniętaZ_7",
                             isReady_filling := "isGotowość_Z_8",
                             isReadyt_emptying := "isGotowość_Z_7",
                             activTank := "Zmienne_sterujące_zbiorników".Zbiornik_4.active_Zb,
                             isAut_Valve_Filling := "Hbit_Auto_Manu_Z8",
                             isAut_Valve_Empting := "Hbit_Auto_Manu_Z7",
                             is_min_Float := "Zmienne_sterujące_zbiorników".Zbiornik_4.is_min_float_Zb,
                             is_max_Float := "Zmienne_sterujące_zbiorników".Zbiornik_4.is_max_float_Zb,
                             isAlarmNinimum_barB5 := "setAlarmNiskie_magistrala",
                             resetAlarmMinimum_barB5 := "resetAlarmNiskie_magistrala",
                             setTank_Work_daily := "DB10_instance_SCADA".TrybSterowania = 1,
                             setTank_Work_selective := "DB10_instance_SCADA".TrybSterowania = 2,
                             setControl_alarm_B5 := "setControl_alarm_B5",
                             set_HWork_tank := "set_HWork_Tank_4",
                             isFilling := "Zmienne_sterujące_zbiorników".Zbiornik_4.isFilling_Zb,
                             isEptying := "Zmienne_sterujące_zbiorników".Zbiornik_4.isEptying_Zb,
                             memRisingLevel_min := "Zmienne_sterujące_zbiorników".Zbiornik_4.memRisingLevel_min_Zb,
                             memRisingLevel_max := "Zmienne_sterujące_zbiorników".Zbiornik_4.memRisingLevel_max_Zb,
                             isLevelMax := "Zmienne_sterujące_zbiorników".Zbiornik_4.isLevelMax_Zb,
                             isLevelMin := "Zmienne_sterujące_zbiorników".Zbiornik_4.isLevelMin_Zb,
                             blok_tank := "Parametryzacja"."Time Tanks".Tank_bocking.blocing_tank4,
                             setSVMO_Z_Wlot => "setSVMO_Z_8",
                             setSVMC_Z_Wlot => "setSVMC_Z_8",
                             setSVMO_Z_Spust => "setSVMO_Z_7",
                             setSVMC_Z_Spust => "setSVMC_Z_7",
                             infoFiling_to_HMI => "HMI.Filing4");
   END_IF;
END_REGION

REGION Network 45: Sterowanie zasuwą Z9 odpływu do pompowni
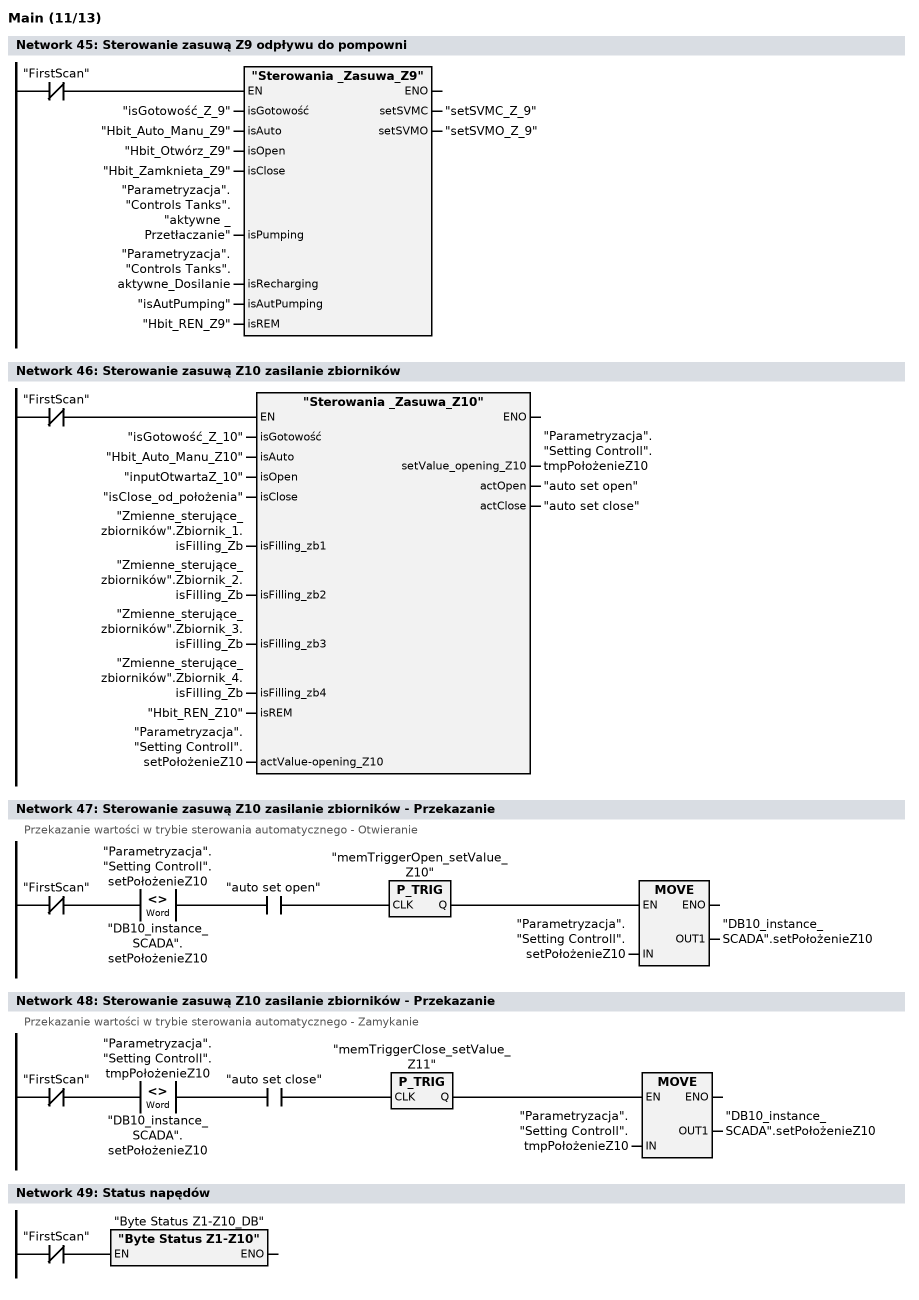
   RUNG wire#powerrail
      I_Contact( "FirstScan" )
      "Sterowania _Zasuwa_Z9"(isGotowość := "isGotowość_Z_9", isAuto := "Hbit_Auto_Manu_Z9", isOpen := "Hbit_Otwórz_Z9", isClose := "Hbit_Zamknieta_Z9", isPumping := "Parametryzacja"."Controls Tanks"."aktywne _Przetłaczanie", isRecharging := "Parametryzacja"."Controls Tanks".aktywne_Dosilanie, isAutPumping := "isAutPumping", isREM := "Hbit_REN_Z9", setSVMC => "setSVMC_Z_9", setSVMO => "setSVMO_Z_9")
   END_RUNG
   // the same network as SCL:
   IF NOT "FirstScan" THEN
       "Sterowania _Zasuwa_Z9"(isGotowość := "isGotowość_Z_9",
                               isAuto := "Hbit_Auto_Manu_Z9",
                               isOpen := "Hbit_Otwórz_Z9",
                               isClose := "Hbit_Zamknieta_Z9",
                               isPumping := "Parametryzacja"."Controls Tanks"."aktywne _Przetłaczanie",
                               isRecharging := "Parametryzacja"."Controls Tanks".aktywne_Dosilanie,
                               isAutPumping := "isAutPumping",
                               isREM := "Hbit_REN_Z9",
                               setSVMC => "setSVMC_Z_9",
                               setSVMO => "setSVMO_Z_9");
   END_IF;
END_REGION

REGION Network 46: Sterowanie zasuwą Z10 zasilanie zbiorników
   RUNG wire#powerrail
      I_Contact( "FirstScan" )
      "Sterowania _Zasuwa_Z10"(isGotowość := "isGotowość_Z_10", isAuto := "Hbit_Auto_Manu_Z10", isOpen := "inputOtwartaZ_10", isClose := "isClose_od_położenia", isFilling_zb1 := "Zmienne_sterujące_zbiorników".Zbiornik_1.isFilling_Zb, isFilling_zb2 := "Zmienne_sterujące_zbiorników".Zbiornik_2.isFilling_Zb, isFilling_zb3 := "Zmienne_sterujące_zbiorników".Zbiornik_3.isFilling_Zb, isFilling_zb4 := "Zmienne_sterujące_zbiorników".Zbiornik_4.isFilling_Zb, isREM := "Hbit_REN_Z10", "actValue-opening_Z10" := "Parametryzacja"."Setting Controll".setPołożenieZ10, setValue_opening_Z10 => "Parametryzacja"."Setting Controll".tmpPołożenieZ10, actOpen => "auto set open", actClose => "auto set close")
   END_RUNG
   // the same network as SCL:
   IF NOT "FirstScan" THEN
       "Sterowania _Zasuwa_Z10"(isGotowość := "isGotowość_Z_10",
                               isAuto := "Hbit_Auto_Manu_Z10",
                               isOpen := "inputOtwartaZ_10",
                               isClose := "isClose_od_położenia",
                               isFilling_zb1 := "Zmienne_sterujące_zbiorników".Zbiornik_1.isFilling_Zb,
                               isFilling_zb2 := "Zmienne_sterujące_zbiorników".Zbiornik_2.isFilling_Zb,
                               isFilling_zb3 := "Zmienne_sterujące_zbiorników".Zbiornik_3.isFilling_Zb,
                               isFilling_zb4 := "Zmienne_sterujące_zbiorników".Zbiornik_4.isFilling_Zb,
                               isREM := "Hbit_REN_Z10",
                               "actValue-opening_Z10" := "Parametryzacja"."Setting Controll".setPołożenieZ10,
                               setValue_opening_Z10 => "Parametryzacja"."Setting Controll".tmpPołożenieZ10,
                               actOpen => "auto set open",
                               actClose => "auto set close");
   END_IF;
END_REGION

REGION Network 47: Sterowanie zasuwą Z10 zasilanie zbiorników - Przekazanie
   // Przekazanie wartości w trybie sterowania automatycznego - Otwieranie
   RUNG wire#powerrail
      I_Contact( "FirstScan" )
      { S7_Templates := "SrcType := Word" } NE_Contact(in1 := "Parametryzacja"."Setting Controll".setPołożenieZ10, in2 := "DB10_instance_SCADA".setPołożenieZ10)
      Contact( "auto set open" )
      P_Trig( "memTriggerOpen_setValue_Z10" )
      Move(in := "Parametryzacja"."Setting Controll".setPołożenieZ10, out1 => "DB10_instance_SCADA".setPołożenieZ10)
   END_RUNG
   // the same network as SCL:
   #_w1 := NOT "FirstScan" AND ("Parametryzacja"."Setting Controll".setPołożenieZ10 <> "DB10_instance_SCADA".setPołożenieZ10) AND "auto set open";
   #_w2 := #_w1 AND NOT "memTriggerOpen_setValue_Z10";   // rising edge
   "memTriggerOpen_setValue_Z10" := #_w1;
   IF #_w2 THEN
       "DB10_instance_SCADA".setPołożenieZ10 := "Parametryzacja"."Setting Controll".setPołożenieZ10;
   END_IF;
END_REGION

REGION Network 48: Sterowanie zasuwą Z10 zasilanie zbiorników - Przekazanie
   // Przekazanie wartości w trybie sterowania automatycznego - Zamykanie
   RUNG wire#powerrail
      I_Contact( "FirstScan" )
      { S7_Templates := "SrcType := Word" } NE_Contact(in1 := "Parametryzacja"."Setting Controll".tmpPołożenieZ10, in2 := "DB10_instance_SCADA".setPołożenieZ10)
      Contact( "auto set close" )
      P_Trig( "memTriggerClose_setValue_Z11" )
      Move(in := "Parametryzacja"."Setting Controll".tmpPołożenieZ10, out1 => "DB10_instance_SCADA".setPołożenieZ10)
   END_RUNG
   // the same network as SCL:
   #_w1 := NOT "FirstScan" AND ("Parametryzacja"."Setting Controll".tmpPołożenieZ10 <> "DB10_instance_SCADA".setPołożenieZ10) AND "auto set close";
   #_w2 := #_w1 AND NOT "memTriggerClose_setValue_Z11";   // rising edge
   "memTriggerClose_setValue_Z11" := #_w1;
   IF #_w2 THEN
       "DB10_instance_SCADA".setPołożenieZ10 := "Parametryzacja"."Setting Controll".tmpPołożenieZ10;
   END_IF;
END_REGION

REGION Network 49: Status napędów
   RUNG wire#powerrail
      I_Contact( "FirstScan" )
      "Byte Status Z1-Z10_DB"()
   END_RUNG
   // the same network as SCL:
   IF NOT "FirstScan" THEN
       "Byte Status Z1-Z10_DB"();   // "Byte Status Z1-Z10"
   END_IF;
END_REGION

REGION Network 50: Kontrola styków momentowych
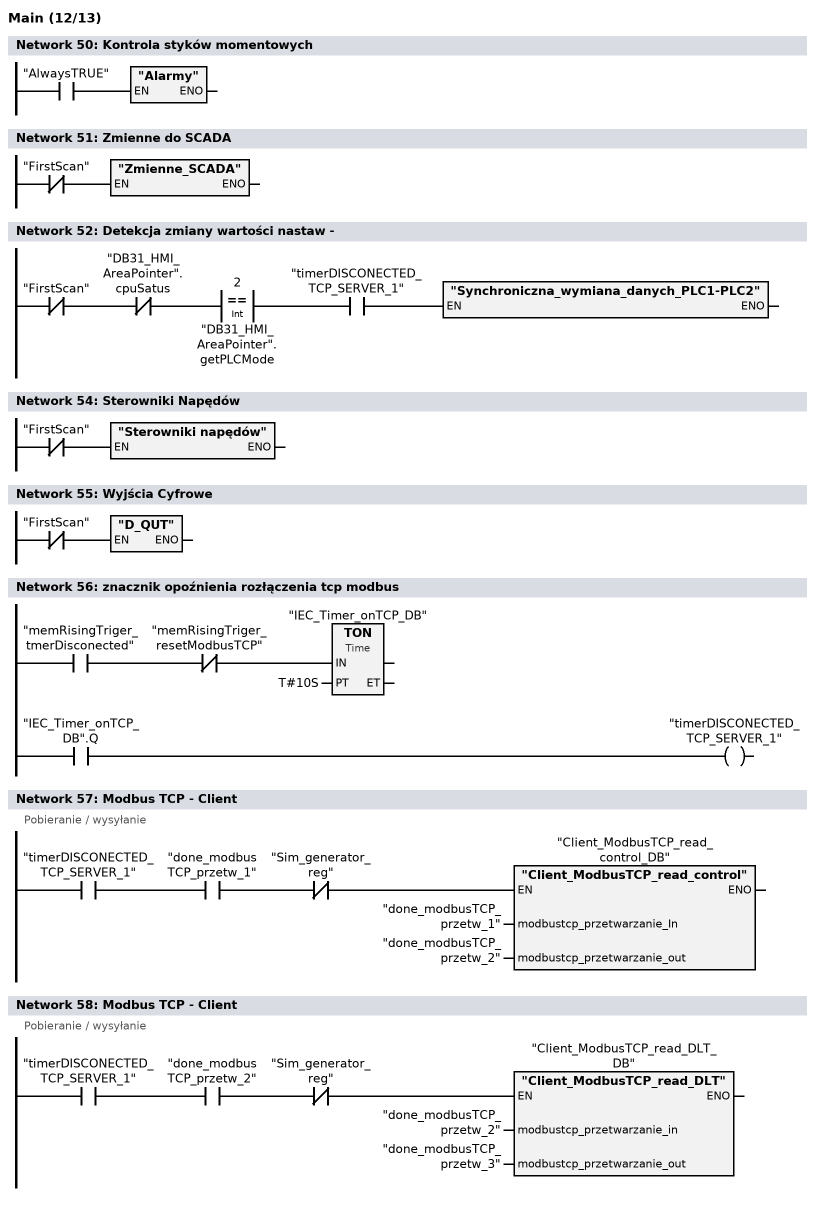
   RUNG wire#powerrail
      Contact( "AlwaysTRUE" )
      "Alarmy"()
   END_RUNG
   // the same network as SCL:
   IF "AlwaysTRUE" THEN "Alarmy"(); END_IF;
END_REGION

REGION Network 51: Zmienne do SCADA
   RUNG wire#powerrail
      I_Contact( "FirstScan" )
      "Zmienne_SCADA"()
   END_RUNG
   // the same network as SCL:
   IF NOT "FirstScan" THEN "Zmienne_SCADA"(); END_IF;
END_REGION

REGION Network 52: Detekcja zmiany wartości nastaw -
   RUNG wire#powerrail
      I_Contact( "FirstScan" )
      I_Contact( "DB31_HMI_AreaPointer".cpuSatus )
      { S7_Templates := "SrcType := Int" } EQ_Contact(in1 := 2, in2 := "DB31_HMI_AreaPointer".getPLCMode)
      Contact( "timerDISCONECTED_TCP_SERVER_1" )
      "Synchroniczna_wymiana_danych_PLC1-PLC2"()
   END_RUNG
   // the same network as SCL:
   IF NOT "FirstScan" AND NOT "DB31_HMI_AreaPointer".cpuSatus AND (2 = "DB31_HMI_AreaPointer".getPLCMode) AND "timerDISCONECTED_TCP_SERVER_1" THEN
       "Synchroniczna_wymiana_danych_PLC1-PLC2"();
   END_IF;
END_REGION

REGION Network 53
   // Funkcja po przeprowadzeniu sprawdzenia czy nastąpiły zmiany w danych przekazuje nowe wartości
END_REGION

REGION Network 54: Sterowniki Napędów
   RUNG wire#powerrail
      I_Contact( "FirstScan" )
      "Sterowniki napędów"()
   END_RUNG
   // the same network as SCL:
   IF NOT "FirstScan" THEN "Sterowniki napędów"(); END_IF;
END_REGION

REGION Network 55: Wyjścia Cyfrowe
   RUNG wire#powerrail
      I_Contact( "FirstScan" )
      "D_QUT"()
   END_RUNG
   // the same network as SCL:
   IF NOT "FirstScan" THEN "D_QUT"(); END_IF;
END_REGION

REGION Network 56: znacznik opoźnienia rozłączenia tcp modbus
   RUNG wire#powerrail
      Contact( "memRisingTriger_tmerDisconected" )
      I_Contact( "memRisingTriger_resetModbusTCP" )
      { S7_Templates := "time_type := Time" } "IEC_Timer_onTCP_DB".TON(pt := T#10S, et =>)
   END_RUNG
   RUNG wire#powerrail
      Contact( "IEC_Timer_onTCP_DB".Q )
      Coil( "timerDISCONECTED_TCP_SERVER_1" )
   END_RUNG
   // the same network as SCL:
   "IEC_Timer_onTCP_DB".TON(IN := "memRisingTriger_tmerDisconected" AND NOT "memRisingTriger_resetModbusTCP",
                           PT := T#10S);
   "timerDISCONECTED_TCP_SERVER_1" := "IEC_Timer_onTCP_DB".Q;
END_REGION

REGION Network 57: Modbus TCP - Client
   // Pobieranie / wysyłanie
   RUNG wire#powerrail
      Contact( "timerDISCONECTED_TCP_SERVER_1" )
      Contact( "done_modbusTCP_przetw_1" )
      I_Contact( "Sim_generator_reg" )
      "Client_ModbusTCP_read_control_DB"(modbustcp_przetwarzanie_In := "done_modbusTCP_przetw_1", modbustcp_przetwarzanie_out := "done_modbusTCP_przetw_2")
   END_RUNG
   // the same network as SCL:
   IF "timerDISCONECTED_TCP_SERVER_1" AND "done_modbusTCP_przetw_1" AND NOT "Sim_generator_reg" THEN
       "Client_ModbusTCP_read_control_DB"(modbustcp_przetwarzanie_In := "done_modbusTCP_przetw_1",   // "Client_ModbusTCP_read_control"
                               modbustcp_przetwarzanie_out := "done_modbusTCP_przetw_2");
   END_IF;
END_REGION

REGION Network 58: Modbus TCP - Client
   // Pobieranie / wysyłanie
   RUNG wire#powerrail
      Contact( "timerDISCONECTED_TCP_SERVER_1" )
      Contact( "done_modbusTCP_przetw_2" )
      I_Contact( "Sim_generator_reg" )
      "Client_ModbusTCP_read_DLT_DB"(modbustcp_przetwarzanie_in := "done_modbusTCP_przetw_2", modbustcp_przetwarzanie_out := "done_modbusTCP_przetw_3")
   END_RUNG
   // the same network as SCL:
   IF "timerDISCONECTED_TCP_SERVER_1" AND "done_modbusTCP_przetw_2" AND NOT "Sim_generator_reg" THEN
       "Client_ModbusTCP_read_DLT_DB"(modbustcp_przetwarzanie_in := "done_modbusTCP_przetw_2",   // "Client_ModbusTCP_read_DLT"
                               modbustcp_przetwarzanie_out := "done_modbusTCP_przetw_3");
   END_IF;
END_REGION

REGION Network 59: Modbus TCP - Client
   // Pobieranie / wysyłanie
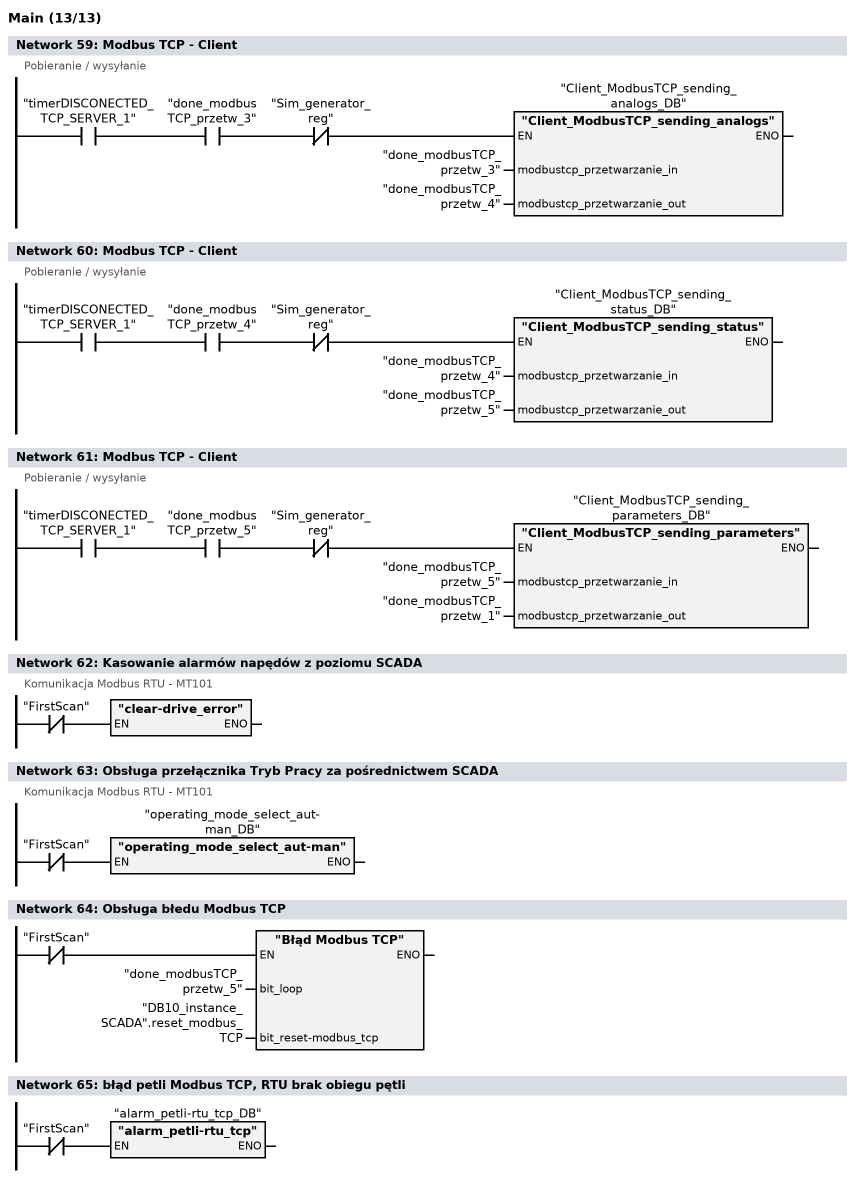
   RUNG wire#powerrail
      Contact( "timerDISCONECTED_TCP_SERVER_1" )
      Contact( "done_modbusTCP_przetw_3" )
      I_Contact( "Sim_generator_reg" )
      "Client_ModbusTCP_sending_analogs_DB"(modbustcp_przetwarzanie_in := "done_modbusTCP_przetw_3", modbustcp_przetwarzanie_out := "done_modbusTCP_przetw_4")
   END_RUNG
   // the same network as SCL:
   IF "timerDISCONECTED_TCP_SERVER_1" AND "done_modbusTCP_przetw_3" AND NOT "Sim_generator_reg" THEN
       "Client_ModbusTCP_sending_analogs_DB"(modbustcp_przetwarzanie_in := "done_modbusTCP_przetw_3",   // "Client_ModbusTCP_sending_analogs"
                               modbustcp_przetwarzanie_out := "done_modbusTCP_przetw_4");
   END_IF;
END_REGION

REGION Network 60: Modbus TCP - Client
   // Pobieranie / wysyłanie
   RUNG wire#powerrail
      Contact( "timerDISCONECTED_TCP_SERVER_1" )
      Contact( "done_modbusTCP_przetw_4" )
      I_Contact( "Sim_generator_reg" )
      "Client_ModbusTCP_sending_status_DB"(modbustcp_przetwarzanie_in := "done_modbusTCP_przetw_4", modbustcp_przetwarzanie_out := "done_modbusTCP_przetw_5")
   END_RUNG
   // the same network as SCL:
   IF "timerDISCONECTED_TCP_SERVER_1" AND "done_modbusTCP_przetw_4" AND NOT "Sim_generator_reg" THEN
       "Client_ModbusTCP_sending_status_DB"(modbustcp_przetwarzanie_in := "done_modbusTCP_przetw_4",   // "Client_ModbusTCP_sending_status"
                               modbustcp_przetwarzanie_out := "done_modbusTCP_przetw_5");
   END_IF;
END_REGION

REGION Network 61: Modbus TCP - Client
   // Pobieranie / wysyłanie
   RUNG wire#powerrail
      Contact( "timerDISCONECTED_TCP_SERVER_1" )
      Contact( "done_modbusTCP_przetw_5" )
      I_Contact( "Sim_generator_reg" )
      "Client_ModbusTCP_sending_parameters_DB"(modbustcp_przetwarzanie_in := "done_modbusTCP_przetw_5", modbustcp_przetwarzanie_out := "done_modbusTCP_przetw_1")
   END_RUNG
   // the same network as SCL:
   IF "timerDISCONECTED_TCP_SERVER_1" AND "done_modbusTCP_przetw_5" AND NOT "Sim_generator_reg" THEN
       "Client_ModbusTCP_sending_parameters_DB"(modbustcp_przetwarzanie_in := "done_modbusTCP_przetw_5",   // "Client_ModbusTCP_sending_parameters"
                               modbustcp_przetwarzanie_out := "done_modbusTCP_przetw_1");
   END_IF;
END_REGION

REGION Network 62: Kasowanie alarmów napędów z poziomu SCADA
   // Komunikacja Modbus RTU - MT101
   RUNG wire#powerrail
      I_Contact( "FirstScan" )
      "clear-drive_error"()
   END_RUNG
   // the same network as SCL:
   IF NOT "FirstScan" THEN "clear-drive_error"(); END_IF;
END_REGION

REGION Network 63: Obsługa przełącznika Tryb Pracy za pośrednictwem SCADA
   // Komunikacja Modbus RTU - MT101
   RUNG wire#powerrail
      I_Contact( "FirstScan" )
      "operating_mode_select_aut-man_DB"()
   END_RUNG
   // the same network as SCL:
   IF NOT "FirstScan" THEN
       "operating_mode_select_aut-man_DB"();   // "operating_mode_select_aut-man"
   END_IF;
END_REGION

REGION Network 64: Obsługa błedu Modbus TCP
   RUNG wire#powerrail
      I_Contact( "FirstScan" )
      "Błąd Modbus TCP"(bit_loop := "done_modbusTCP_przetw_5", "bit_reset-modbus_tcp" := "DB10_instance_SCADA".reset_modbus_TCP)
   END_RUNG
   // the same network as SCL:
   IF NOT "FirstScan" THEN
       "Błąd Modbus TCP"(bit_loop := "done_modbusTCP_przetw_5",
                         "bit_reset-modbus_tcp" := "DB10_instance_SCADA".reset_modbus_TCP);
   END_IF;
END_REGION

REGION Network 65: błąd petli Modbus TCP, RTU brak obiegu pętli
   RUNG wire#powerrail
      I_Contact( "FirstScan" )
      "alarm_petli-rtu_tcp_DB"()
   END_RUNG
   // the same network as SCL:
   IF NOT "FirstScan" THEN
       "alarm_petli-rtu_tcp_DB"();   // "alarm_petli-rtu_tcp"
   END_IF;
END_REGION
END_ORGANIZATION_BLOCK
